# B&R Automation Studio project Assembly_and_ST
Automation Studio 4.5.2.102; technology packages: mappCockpit 5.7.0, mappMotion 5.7.1, mappView 5.7.1

## Configuration Config1

CPU 5PC900.TS77-04, AutomationRuntime D4.52, Build 4.1.2, Vc V4.52.0

### Task classes (Cpu.sw)
```
Cyclic#1 (cycle 800 us, tolerance 0 us):
  ST_Main <- SuperTrak_Module.ST_Main.prg
  MainContro <- Assembly_Module.MainControl.prg
Cyclic#2 (cycle 1600 us, tolerance 0 us):
  AlarmHandl <- Events_handling.AlarmHandling.prg
  AssemblyIn <- Assembly_Module.AssemblyInterface.prg
Cyclic#3 (cycle 9600 us, tolerance 9600 us):
  DisableBra <- Assembly_Module.DisableBrake.prg
  StateMachi <- SuperTrak_Module.StateMachine_SuperTrak.prg
Cyclic#4 (cycle 49600 us, tolerance 49600 us):
  ST_Visu <- SuperTrak_Module.ST_Visu.prg
  EventLogge <- Events_handling.EventLoggerMNG.prg
DataObjects: McAcpSys
Binaries: mvLoader, arcoal, McMechSys, arflatprv, arsvcreg, McProfGen, TCData, McPathXT, mCoWebSc, McAcpSim, McAcpDrv, udbdef, TCLang, Settings, iomap, Config_2, Hierarchy, Config_4, sysconf, ashwac, Config_1, ashwd, asfw, User, arconfig, Config_3, Role, OpcUaMap
Libraries: DataObj, AsArLog, sys_lib, FileIO, AsArProf, AsMem, brsystem, NcGlobal, runtime, astime, AsBrMath, StCom, SuperTrak, AsIecCon, AsBrStr, standard, ArEventLog, AsIODiag, AsGuard, AsTCP, AsIOTime, MpTool, MpBase, McAxGroup, McBase, MpRobotics, MpCnc, MpAxis, McAxis, McProgInt, McPathGen, McPureVAx, McDS402Ax, McAcpPar, McAcpAx, CoTrace, AsZip, asstring, AsARCfg, MpServer, aspciext, asepl, powerlnk, aruser
```

### Hardware
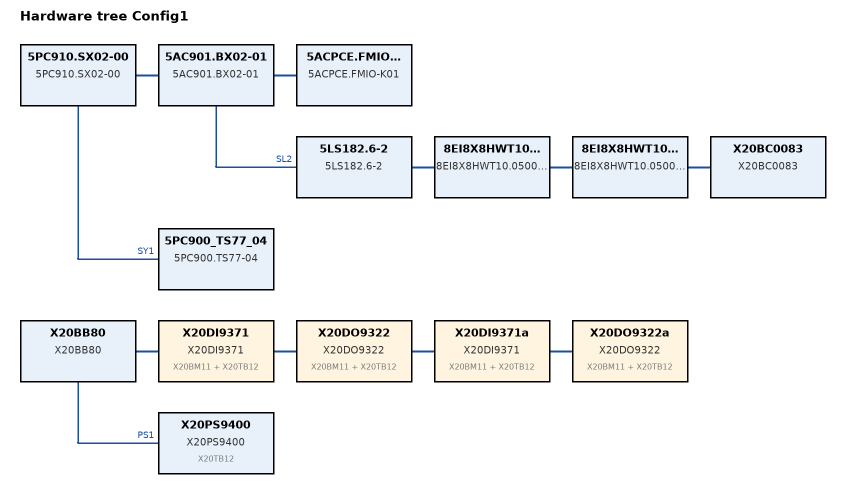
```
5AC901.BX02-01 : 5AC901.BX02-01 v1.1.1.0  [SY -> 5PC910.SX02-00.SY3]
5ACPCE.FMIO-K01 : 5ACPCE.FMIO-K01 v1.0.6.0  [SL -> 5AC901.BX02-01.SL1]
5LS182.6-2 : 5LS182.6-2 v1.3.1.0  [SL -> 5AC901.BX02-01.SL2]
  Connector IF1:
    CycleTime = 800
    Channel1
    ChannelID1 = McAcpBroadcast
    ChannelType1 = OCTET[96]
5PC900_TS77_04 : 5PC900.TS77-04 v2.0.0.0  [SY -> 5PC910.SX02-00.SY1]
  ConfigurationID = ygc_Config1
  UserPartitionSize = 14
  SimulationIPAddress = 192.168.0.101
  UserRamDevice = PCI.2.LS182.SRAM
  UserRamSize = 100000
  RemMemDevice = PCI.2.LS182.SRAM
  RemMemSize = 2048
  PermanentPvSize = 512
  RemanentGlobalPvSize = 512
  VolatileGlobalPvSize = 1026080
  SystemLoggerSize = 614400
  UserLoggerSize = 614400
  TimerDeviceType = EPLX2X
  TimerDevice = 5LS182.6-2.IF1
  TaskClassIdleTime = 800
  Cyclic1Duration = 800
  Cyclic1Tolerance = 0
  Cyclic2Duration = 1600
  Cyclic2Tolerance = 0
  Cyclic3Duration = 9600
  Cyclic3Tolerance = 9600
  Cyclic4Duration = 49600
  Cyclic4Tolerance = 49600
  Cyclic8Duration = 9600
  Cyclic8Tolerance = 0
  FtpUser1
  FtpUsername1 = itq
  FtpUserPassword1 = 7p7ZSnRe8FOUJ14P8lbKBhjsJ4NWIj5puPFWROWS8Pg=
  FtpUserSalt1 = MjfVbkzs
  FTPAccessRight1 = 0
  ActivateOpcUa = 1
  OpcUa_AuthenticationSecurityPolicy_EnableNone = 1
  OpcUa_AuthenticationSecurityPolicy_EnableBasic128Rsa15 = 1
  OpcUaInformationModels_PV_Version = 1
5PC910.SX02-00 : 5PC910.SX02-00 v2.0.0.0
  Connector IF1:
    AssignedOperatingSystem = ARemb
  Connector IF3:
    AssignedOperatingSystem = ARemb
    ActivateDevice = 1
    Mode = Manual
    InternetAddress = 192.168.0.5
    SubnetMask = 255.255.255.0
  Connector IF4:
    AssignedOperatingSystem = ARemb
    ActivateDevice = 1
  Connector IF5:
    AssignedOperatingSystem = ARemb
  Connector IF6:
    AssignedOperatingSystem = ARemb
  Connector IF7:
    AssignedOperatingSystem = ARemb
  Connector IF8:
    AssignedOperatingSystem = ARemb
  Connector IF9:
    AssignedOperatingSystem = ARemb
8EI8X8HWT10.0500-1 : 8EI8X8HWT10.0500-1 v2.2.0.0  [PLK1 -> 5LS182.6-2.IF1 [Cable Type=PowerlinkCable, Length=10, Version=1.0.0.2]; PLK2 -> 8EI8X8HWT10.0500-1a.PLK1 [Cable Type=PowerlinkCable, Length=10, Version=1.0.0.2]]
  DriveConfiguration/Module:
    McAcoposTypeID = AcoposP3TConfig
    ActivateACOPOSSimulationOnPLC = 0
  DriveConfiguration/Encoder/EncoderX41:
    InterfaceType = EnDat
  DriveConfiguration/Encoder/EncoderX42:
    InterfaceType = EnDat
  DriveConfiguration/Encoder/EncoderX43:
    InterfaceType = EnDat
  DriveConfiguration/Channel[1]:
    License = 1
  DriveConfiguration/Channel[1]/RealAxis:
    AxisReference = gAxisQ1
  DriveConfiguration/Channel[1]/RealAxis/MechanicalElements/Gearbox:
    InputIsReadOnly = 1
    Input = 81818
    OutputIsReadOnly = 1
    Output = 1000
  DriveConfiguration/Channel[1]/RealAxis/MechanicalElements/RotaryToLinearTransformation:
    ReferenceDistanceIsReadOnly = 1
    ReferenceDistance = 360
  DriveConfiguration/Channel[1]/RealAxis/Controller:
    ModeIsReadOnly = 1
    Mode = PositionControllerWithTorqueFeedForward
  DriveConfiguration/Channel[1]/RealAxis/Controller/Mode/Position:
    ProportionalGainIsReadOnly = 1
    ProportionalGain = 75.0
    IntegrationTimeIsReadOnly = 1
    IntegrationTime = 0.0
    TotalDelayTime = 0.0004
  DriveConfiguration/Channel[1]/RealAxis/Controller/Mode/Speed:
    ProportionalGainIsReadOnly = 1
    ProportionalGain = 2.0
    IntegrationTimeIsReadOnly = 1
    IntegrationTime = 0.0
    FilterTimeIsReadOnly = 1
    FilterTime = 0.0008
  DriveConfiguration/Channel[1]/RealAxis/Controller/Mode:
    FeedForwardIsReadOnly = 1
    FeedForward = CyclicValueFromAxesGroup
  DriveConfiguration/Channel[1]/RealAxis/Controller/Mode/LoopFilters:
    LoopFilter1 = NotUsed
    LoopFilter2 = NotUsed
    LoopFilter3 = NotUsed
  DriveConfiguration/Channel[1]/RealAxis/Homing:
    Mode = RestorePosition
    RestorePositionVariable = ::MainContro:ResPos[0]
  DriveConfiguration/Channel[1]/RealAxis/StopReaction:
    Quickstop = DecelerationLimit
    DriveError = DecelerationLimit
  DriveConfiguration/Channel[1]/RealAxis/MovementErrorLimits:
    PositionError = 1.0
    VelocityErrorMonitoring = Automatic1
  DriveConfiguration/Channel[1]/RealAxis:
    JerkFilter = Used
  DriveConfiguration/Channel[1]/RealAxis/JerkFilter:
    JerkTime = 0.01
  DriveConfiguration/Channel[1]/RealAxis/DigitalInputs/HomingSwitch:
    Source = NotUsed
    Level = High
  DriveConfiguration/Channel[1]/RealAxis/DigitalInputs/PositiveLimitSwitch:
    Source = NotUsed
    Level = High
  DriveConfiguration/Channel[1]/RealAxis/DigitalInputs/NegativeLimitSwitch:
    Source = NotUsed
    Level = High
  DriveConfiguration/Channel[1]/RealAxis/DigitalInputs/Trigger1:
    Source = X8Trigger1
    Level = High
  DriveConfiguration/Channel[1]/RealAxis/DigitalInputs/Trigger2:
    Source = X8Trigger2
    Level = High
  DriveConfiguration/Channel[1]/RealAxis/DigitalInputs/Quickstop:
    Input = Trigger2
  DriveConfiguration/Channel[1]/RealAxis/Simulation:
    SimulationModeOnPLC = SetValueGeneration
    SimulationModeOnACOPOS = NotUsed
  DriveConfiguration/Channel[2]:
    License = 1
  DriveConfiguration/Channel[2]/RealAxis:
    AxisReference = gAxisQ3
  DriveConfiguration/Channel[2]/RealAxis/MechanicalElements/Gearbox:
    InputIsReadOnly = 1
    Input = 72
    OutputIsReadOnly = 1
    Output = 1
  DriveConfiguration/Channel[2]/RealAxis/MechanicalElements/RotaryToLinearTransformation:
    ReferenceDistanceIsReadOnly = 1
    ReferenceDistance = 360
  DriveConfiguration/Channel[2]/RealAxis/Controller:
    ModeIsReadOnly = 1
    Mode = PositionControllerWithTorqueFeedForward
  DriveConfiguration/Channel[2]/RealAxis/Controller/Mode/Position:
    ProportionalGainIsReadOnly = 1
    ProportionalGain = 50.0
    IntegrationTimeIsReadOnly = 1
    IntegrationTime = 0.0
    TotalDelayTime = 0.0004
  DriveConfiguration/Channel[2]/RealAxis/Controller/Mode/Speed:
    ProportionalGainIsReadOnly = 1
    ProportionalGain = 1.5
    IntegrationTimeIsReadOnly = 1
    IntegrationTime = 0.0
    FilterTimeIsReadOnly = 1
    FilterTime = 0.0008
  DriveConfiguration/Channel[2]/RealAxis/Controller/Mode:
    FeedForwardIsReadOnly = 1
    FeedForward = CyclicValueFromAxesGroup
  DriveConfiguration/Channel[2]/RealAxis/Controller/Mode/LoopFilters:
    LoopFilter1 = NotUsed
    LoopFilter2 = NotUsed
    LoopFilter3 = NotUsed
  DriveConfiguration/Channel[2]/RealAxis/Homing:
    Mode = RestorePosition
    RestorePositionVariable = ::MainContro:ResPos[2]
  DriveConfiguration/Channel[2]/RealAxis/StopReaction:
    Quickstop = DecelerationLimit
    DriveError = DecelerationLimit
  DriveConfiguration/Channel[2]/RealAxis/MovementErrorLimits:
    PositionError = 1.0
    VelocityErrorMonitoring = Automatic1
  DriveConfiguration/Channel[2]/RealAxis:
    JerkFilter = Used
  DriveConfiguration/Channel[2]/RealAxis/JerkFilter:
    JerkTime = 0.01
  DriveConfiguration/Channel[2]/RealAxis/DigitalInputs/HomingSwitch:
    Source = NotUsed
    Level = High
  DriveConfiguration/Channel[2]/RealAxis/DigitalInputs/PositiveLimitSwitch:
    Source = NotUsed
    Level = High
  DriveConfiguration/Channel[2]/RealAxis/DigitalInputs/NegativeLimitSwitch:
    Source = NotUsed
    Level = High
  DriveConfiguration/Channel[2]/RealAxis/DigitalInputs/Trigger1:
    Source = X8Trigger1
    Level = High
  DriveConfiguration/Channel[2]/RealAxis/DigitalInputs/Trigger2:
    Source = X8Trigger2
    Level = High
  DriveConfiguration/Channel[2]/RealAxis/DigitalInputs/Quickstop:
    Input = Trigger2
  DriveConfiguration/Channel[2]/RealAxis/Simulation:
    SimulationModeOnPLC = SetValueGeneration
    SimulationModeOnACOPOS = NotUsed
  DriveConfiguration/Channel[3]:
    License = 1
  DriveConfiguration/Channel[3]/RealAxis:
    AxisReference = gAxisQ5
  DriveConfiguration/Channel[3]/RealAxis/MechanicalElements/Gearbox:
    InputIsReadOnly = 1
    Input = 612
    OutputIsReadOnly = 1
    Output = 10
  DriveConfiguration/Channel[3]/RealAxis/MechanicalElements/RotaryToLinearTransformation:
    ReferenceDistanceIsReadOnly = 1
    ReferenceDistance = 360
  DriveConfiguration/Channel[3]/RealAxis/Controller:
    ModeIsReadOnly = 1
    Mode = PositionControllerWithTorqueFeedForward
  DriveConfiguration/Channel[3]/RealAxis/Controller/Mode/Position:
    ProportionalGainIsReadOnly = 1
    ProportionalGain = 200.0
    IntegrationTimeIsReadOnly = 1
    IntegrationTime = 0.0
    TotalDelayTime = 0.0004
  DriveConfiguration/Channel[3]/RealAxis/Controller/Mode/Speed:
    ProportionalGainIsReadOnly = 1
    ProportionalGain = 1.5
    IntegrationTimeIsReadOnly = 1
    IntegrationTime = 0.0
    FilterTimeIsReadOnly = 1
    FilterTime = 0.0008
  DriveConfiguration/Channel[3]/RealAxis/Controller/Mode:
    FeedForwardIsReadOnly = 1
    FeedForward = CyclicValueFromAxesGroup
  DriveConfiguration/Channel[3]/RealAxis/Controller/Mode/LoopFilters:
    LoopFilter1 = NotUsed
    LoopFilter2 = NotUsed
    LoopFilter3 = NotUsed
  DriveConfiguration/Channel[3]/RealAxis/Homing:
    Mode = RestorePosition
    RestorePositionVariable = ::MainContro:ResPos[4]
  DriveConfiguration/Channel[3]/RealAxis/StopReaction:
    Quickstop = DecelerationLimit
    DriveError = DecelerationLimit
  DriveConfiguration/Channel[3]/RealAxis/MovementErrorLimits:
    PositionError = 1.0
    VelocityErrorMonitoring = Automatic1
  DriveConfiguration/Channel[3]/RealAxis:
    JerkFilter = Used
  DriveConfiguration/Channel[3]/RealAxis/JerkFilter:
    JerkTime = 0.01
  DriveConfiguration/Channel[3]/RealAxis/DigitalInputs/HomingSwitch:
    Source = NotUsed
    Level = High
  DriveConfiguration/Channel[3]/RealAxis/DigitalInputs/PositiveLimitSwitch:
    Source = NotUsed
    Level = High
  DriveConfiguration/Channel[3]/RealAxis/DigitalInputs/NegativeLimitSwitch:
    Source = NotUsed
    Level = High
  DriveConfiguration/Channel[3]/RealAxis/DigitalInputs/Trigger1:
    Source = X8Trigger1
    Level = High
  DriveConfiguration/Channel[3]/RealAxis/DigitalInputs/Trigger2:
    Source = X8Trigger2
    Level = High
  DriveConfiguration/Channel[3]/RealAxis/DigitalInputs/Quickstop:
    Input = Trigger2
  DriveConfiguration/Channel[3]/RealAxis/Simulation:
    SimulationModeOnPLC = SetValueGeneration
    SimulationModeOnACOPOS = NotUsed
8EI8X8HWT10.0500-1a : 8EI8X8HWT10.0500-1 v2.2.0.0  [PLK1 -> 8EI8X8HWT10.0500-1.PLK2 [Cable Type=PowerlinkCable, Length=10, Version=1.0.0.2]; PLK2 -> X20BC0083.PLK1 [Cable Type=PowerlinkCable, Length=10, Version=1.0.0.2]]
  DriveConfiguration/Module:
    McAcoposTypeID = AcoposP3TConfig
    ActivateACOPOSSimulationOnPLC = 0
  DriveConfiguration/Encoder/EncoderX41:
    InterfaceType = EnDat
  DriveConfiguration/Encoder/EncoderX42:
    InterfaceType = EnDat
  DriveConfiguration/Encoder/EncoderX43:
    InterfaceType = EnDat
  DriveConfiguration/Channel[1]:
    License = 1
  DriveConfiguration/Channel[1]/RealAxis:
    AxisReference = gAxisQ2
  DriveConfiguration/Channel[1]/RealAxis/MechanicalElements/Gearbox:
    InputIsReadOnly = 1
    Input = 80
    OutputIsReadOnly = 1
    Output = 1
  DriveConfiguration/Channel[1]/RealAxis/MechanicalElements/RotaryToLinearTransformation:
    ReferenceDistanceIsReadOnly = 1
    ReferenceDistance = 360
  DriveConfiguration/Channel[1]/RealAxis/Controller:
    ModeIsReadOnly = 1
    Mode = PositionControllerWithTorqueFeedForward
  DriveConfiguration/Channel[1]/RealAxis/Controller/Mode/Position:
    ProportionalGainIsReadOnly = 1
    ProportionalGain = 50.0
    IntegrationTimeIsReadOnly = 1
    IntegrationTime = 0.0
    TotalDelayTime = 0.0004
  DriveConfiguration/Channel[1]/RealAxis/Controller/Mode/Speed:
    ProportionalGainIsReadOnly = 1
    ProportionalGain = 2.0
    IntegrationTimeIsReadOnly = 1
    IntegrationTime = 0.0
    FilterTimeIsReadOnly = 1
    FilterTime = 0.0008
  DriveConfiguration/Channel[1]/RealAxis/Controller/Mode:
    FeedForwardIsReadOnly = 1
    FeedForward = CyclicValueFromAxesGroup
  DriveConfiguration/Channel[1]/RealAxis/Controller/Mode/LoopFilters:
    LoopFilter1 = NotUsed
    LoopFilter2 = NotUsed
    LoopFilter3 = NotUsed
  DriveConfiguration/Channel[1]/RealAxis/Homing:
    Mode = RestorePosition
    RestorePositionVariable = ::MainContro:ResPos[1]
  DriveConfiguration/Channel[1]/RealAxis/StopReaction:
    Quickstop = DecelerationLimit
    DriveError = DecelerationLimit
  DriveConfiguration/Channel[1]/RealAxis/MovementErrorLimits:
    PositionError = 1.0
    VelocityErrorMonitoring = Automatic1
  DriveConfiguration/Channel[1]/RealAxis:
    JerkFilter = Used
  DriveConfiguration/Channel[1]/RealAxis/JerkFilter:
    JerkTime = 0.01
  DriveConfiguration/Channel[1]/RealAxis/DigitalInputs/HomingSwitch:
    Source = NotUsed
    Level = High
  DriveConfiguration/Channel[1]/RealAxis/DigitalInputs/PositiveLimitSwitch:
    Source = NotUsed
    Level = High
  DriveConfiguration/Channel[1]/RealAxis/DigitalInputs/NegativeLimitSwitch:
    Source = NotUsed
    Level = High
  DriveConfiguration/Channel[1]/RealAxis/DigitalInputs/Trigger1:
    Source = X8Trigger1
    Level = High
  DriveConfiguration/Channel[1]/RealAxis/DigitalInputs/Trigger2:
    Source = X8Trigger2
    Level = High
  DriveConfiguration/Channel[1]/RealAxis/DigitalInputs/Quickstop:
    Input = Trigger2
  DriveConfiguration/Channel[1]/RealAxis/Simulation:
    SimulationModeOnPLC = SetValueGeneration
    SimulationModeOnACOPOS = NotUsed
  DriveConfiguration/Channel[2]:
    License = 1
  DriveConfiguration/Channel[2]/RealAxis:
    AxisReference = gAxisQ4
  DriveConfiguration/Channel[2]/RealAxis/MechanicalElements/Gearbox:
    InputIsReadOnly = 1
    Input = 612
    OutputIsReadOnly = 1
    Output = 10
  DriveConfiguration/Channel[2]/RealAxis/MechanicalElements/RotaryToLinearTransformation:
    ReferenceDistanceIsReadOnly = 1
    ReferenceDistance = 360
  DriveConfiguration/Channel[2]/RealAxis/Controller:
    ModeIsReadOnly = 1
    Mode = PositionControllerWithTorqueFeedForward
  DriveConfiguration/Channel[2]/RealAxis/Controller/Mode/Position:
    ProportionalGainIsReadOnly = 1
    ProportionalGain = 100.0
    IntegrationTimeIsReadOnly = 1
    IntegrationTime = 0.0
    TotalDelayTime = 0.0004
  DriveConfiguration/Channel[2]/RealAxis/Controller/Mode/Speed:
    ProportionalGainIsReadOnly = 1
    ProportionalGain = 2.0
    IntegrationTimeIsReadOnly = 1
    IntegrationTime = 0.0
    FilterTimeIsReadOnly = 1
    FilterTime = 0.0008
  DriveConfiguration/Channel[2]/RealAxis/Controller/Mode:
    FeedForwardIsReadOnly = 1
    FeedForward = CyclicValueFromAxesGroup
  DriveConfiguration/Channel[2]/RealAxis/Controller/Mode/LoopFilters:
    LoopFilter1 = NotUsed
    LoopFilter2 = NotUsed
    LoopFilter3 = NotUsed
  DriveConfiguration/Channel[2]/RealAxis/Homing:
    Mode = RestorePosition
    RestorePositionVariable = ::MainContro:ResPos[3]
  DriveConfiguration/Channel[2]/RealAxis/StopReaction:
    Quickstop = DecelerationLimit
    DriveError = DecelerationLimit
  DriveConfiguration/Channel[2]/RealAxis/MovementErrorLimits:
    PositionError = 1.0
    VelocityErrorMonitoring = Automatic1
  DriveConfiguration/Channel[2]/RealAxis:
    JerkFilter = Used
  DriveConfiguration/Channel[2]/RealAxis/JerkFilter:
    JerkTime = 0.01
  DriveConfiguration/Channel[2]/RealAxis/DigitalInputs/HomingSwitch:
    Source = NotUsed
    Level = High
  DriveConfiguration/Channel[2]/RealAxis/DigitalInputs/PositiveLimitSwitch:
    Source = NotUsed
    Level = High
  DriveConfiguration/Channel[2]/RealAxis/DigitalInputs/NegativeLimitSwitch:
    Source = NotUsed
    Level = High
  DriveConfiguration/Channel[2]/RealAxis/DigitalInputs/Trigger1:
    Source = X8Trigger1
    Level = High
  DriveConfiguration/Channel[2]/RealAxis/DigitalInputs/Trigger2:
    Source = X8Trigger2
    Level = High
  DriveConfiguration/Channel[2]/RealAxis/DigitalInputs/Quickstop:
    Input = Trigger2
  DriveConfiguration/Channel[2]/RealAxis/Simulation:
    SimulationModeOnPLC = SetValueGeneration
    SimulationModeOnACOPOS = NotUsed
  DriveConfiguration/Channel[3]:
    License = 1
  DriveConfiguration/Channel[3]/RealAxis:
    AxisReference = gAxisQ6
  DriveConfiguration/Channel[3]/RealAxis/MechanicalElements/Gearbox:
    InputIsReadOnly = 1
    Input = 40
    OutputIsReadOnly = 1
    Output = 1
  DriveConfiguration/Channel[3]/RealAxis/MechanicalElements/RotaryToLinearTransformation:
    ReferenceDistanceIsReadOnly = 1
    ReferenceDistance = 360
  DriveConfiguration/Channel[3]/RealAxis/Controller:
    ModeIsReadOnly = 1
    Mode = PositionControllerWithTorqueFeedForward
  DriveConfiguration/Channel[3]/RealAxis/Controller/Mode/Position:
    ProportionalGainIsReadOnly = 1
    ProportionalGain = 200.0
    IntegrationTimeIsReadOnly = 1
    IntegrationTime = 0.0
    TotalDelayTime = 0.0004
  DriveConfiguration/Channel[3]/RealAxis/Controller/Mode/Speed:
    ProportionalGainIsReadOnly = 1
    ProportionalGain = 1.5
    IntegrationTimeIsReadOnly = 1
    IntegrationTime = 0.0
    FilterTimeIsReadOnly = 1
    FilterTime = 0.0008
  DriveConfiguration/Channel[3]/RealAxis/Controller/Mode:
    FeedForwardIsReadOnly = 1
    FeedForward = CyclicValueFromAxesGroup
  DriveConfiguration/Channel[3]/RealAxis/Controller/Mode/LoopFilters:
    LoopFilter1 = NotUsed
    LoopFilter2 = NotUsed
    LoopFilter3 = NotUsed
  DriveConfiguration/Channel[3]/RealAxis/Homing:
    Mode = RestorePosition
    RestorePositionVariable = ::MainContro:ResPos[5]
  DriveConfiguration/Channel[3]/RealAxis/StopReaction:
    Quickstop = DecelerationLimit
    DriveError = DecelerationLimit
  DriveConfiguration/Channel[3]/RealAxis/MovementErrorLimits:
    PositionError = 1.0
    VelocityErrorMonitoring = Automatic1
  DriveConfiguration/Channel[3]/RealAxis:
    JerkFilter = Used
  DriveConfiguration/Channel[3]/RealAxis/JerkFilter:
    JerkTime = 0.01
  DriveConfiguration/Channel[3]/RealAxis/DigitalInputs/HomingSwitch:
    Source = NotUsed
    Level = High
  DriveConfiguration/Channel[3]/RealAxis/DigitalInputs/PositiveLimitSwitch:
    Source = NotUsed
    Level = High
  DriveConfiguration/Channel[3]/RealAxis/DigitalInputs/NegativeLimitSwitch:
    Source = NotUsed
    Level = High
  DriveConfiguration/Channel[3]/RealAxis/DigitalInputs/Trigger1:
    Source = X8Trigger1
    Level = High
  DriveConfiguration/Channel[3]/RealAxis/DigitalInputs/Trigger2:
    Source = X8Trigger2
    Level = High
  DriveConfiguration/Channel[3]/RealAxis/DigitalInputs/Quickstop:
    Input = Trigger2
  DriveConfiguration/Channel[3]/RealAxis/Simulation:
    SimulationModeOnPLC = SetValueGeneration
    SimulationModeOnACOPOS = NotUsed
X20BB80 : X20BB80 v1.0.2.0
X20BC0083 : X20BC0083 v2.7.0.0  [PLK1 -> 8EI8X8HWT10.0500-1a.PLK2 [Cable Type=PowerlinkCable, Length=10, Version=1.0.0.2]; SL -> X20BB80.SL1]
  Supervision = off
X20BM11 : X20BM11 v1.0.0.1  [X2X1 -> X20BB80.IF1]
X20BM11a : X20BM11 v1.0.0.1  [X2X1 -> X20BM11.X2X2]
X20BM11b : X20BM11 v1.0.0.1  [X2X1 -> X20BM11c.X2X2]
X20BM11c : X20BM11 v1.0.0.1  [X2X1 -> X20BM11a.X2X2]
X20DI9371 : X20DI9371 v1.0.2.0  [SS1 -> X20TB12.SS; SL -> X20BM11.SL1]
  Supervision = off
X20DI9371a : X20DI9371 v1.0.2.0  [SS1 -> X20TB12d.SS; SL -> X20BM11c.SL1]
  Supervision = off
X20DO9322 : X20DO9322 v1.0.3.0  [SS1 -> X20TB12b.SS; SL -> X20BM11a.SL1]
  Supervision = off
X20DO9322a : X20DO9322 v1.0.3.0  [SS1 -> X20TB12c.SS; SL -> X20BM11b.SL1]
  Supervision = off
X20PS9400 : X20PS9400 v1.0.2.4  [SS1 -> X20TB12a.SS; PS -> X20BB80.PS1]
  Supervision = off
X20TB12 : X20TB12 v1.0.0.0
X20TB12a : X20TB12 v1.0.0.0
X20TB12b : X20TB12 v1.0.0.0
X20TB12c : X20TB12 v1.0.0.0
X20TB12d : X20TB12 v1.0.0.0
```

### IoMap.iom - 5PC900_TS77_04/IoMap.iom
```iecst
VAR_CONFIG
	::LED_Green AT %QX."X20DO9322".DigitalOutput06;
	::LED_Blue AT %QX."X20DO9322".DigitalOutput07;
	::LED_Red AT %QX."X20DO9322".DigitalOutput08;
	::QA_Actuator_UP AT %QX."X20DO9322".DigitalOutput09;
	::QA_Actuator_DOWN AT %QX."X20DO9322".DigitalOutput10;
	HW_Comau_Gripper AT %QX."X20DO9322a".DigitalOutput01;
	::HW_Assem_RightDoorSensor AT %IX."X20DI9371a".DigitalInput01;
	::HW_Assem_LeftDoorSensor AT %IX."X20DI9371a".DigitalInput02;
	Cyclic#2.::QA_Door_Closed AT %IX."X20DI9371".DigitalInput01;
	ST_LightBarrier_SecurityOut1_R AT %IX."X20DI9371".DigitalInput03;
	ST_LightBarrier_SecurityOut2_R AT %IX."X20DI9371".DigitalInput02;
	::HW_Assem_PelletPresent AT %IX."X20DI9371".DigitalInput06;
	::HW_Assem_PlasticCupsDrawer AT %IX."X20DI9371".DigitalInput05;
	::HW_Assem_PaperCupsDrawer AT %IX."X20DI9371".DigitalInput04;
	::HW_Assem_PlasticLock AT %QX."X20DO9322".DigitalOutput11;
	::HW_Assem_PaperLock AT %QX."X20DO9322".DigitalOutput12;
	::Outfeed_Full AT %IX."X20DI9371a".DigitalInput04;
	::StateMachi:QA_finished AT %IX."X20DI9371a".DigitalInput07;
	::Outfeed_Actuator_BACK AT %QX."X20DO9322".DigitalOutput01;
	::Outfeed_Actuator_FRONT  AT %QX."X20DO9322".DigitalOutput02;
	::Outfeed_Actuator_UP AT %QX."X20DO9322".DigitalOutput03;
	::Outfeed_Actuator_DOWN AT %QX."X20DO9322".DigitalOutput04;
	::Outfeed_LED_Blue  AT %QX."X20DO9322a".DigitalOutput02;
	::Outfeed_LED_Red AT %QX."X20DO9322a".DigitalOutput03;
	::Outfeed_LED_Green AT %QX."X20DO9322a".DigitalOutput04;
END_VAR
```

### Config_3.mechanicalsystem - 5PC900_TS77_04/mappMotion/ComauRacer3/Config_3.mechanicalsystem
```
Element MechSys_ComauRacer3 (Type=mechanicalsystem)
  Type = 6AxesRoboarm
    Subtype = 6AxesRoboarmB
      Description = Standard
        Dimensions:
          TranslationFromBaseToQ1IsReadOnly = 1
          TranslationFromBaseToQ1:
            X = 0.0
            Y = 0.0
            Z = 0.0
          TranslationFromQ1ToQ2IsReadOnly = 1
          TranslationFromQ1ToQ2:
            X = 50.0
            Y = 0.0
            Z = 365.0
          TranslationFromQ2ToQ3IsReadOnly = 1
          TranslationFromQ2ToQ3:
            X = 0.0
            Y = 0.0
            Z = 270.0
          TranslationFromQ3ToQ4IsReadOnly = 1
          TranslationFromQ3ToQ4:
            X = -50.0
            Y = 0.0
            Z = 0.0
          TranslationFromQ4ToQ5IsReadOnly = 1
          TranslationFromQ4ToQ5:
            Z = 305.94
          TranslationFromQ5ToQ6IsReadOnly = 1
          TranslationFromQ5ToQ6:
            Z = 0.0
          TranslationFromQ6ToFlange:
            X = 0.0
            Y = 0.0
            Z = 255
        Offsets:
          JointAxisIsReadOnly = 1
          JointAxis[1] = 0.0
          JointAxis[2] = 0.0
          JointAxis[3] = 0.0
          JointAxis[4] = 0.0
          JointAxis[5] = 0.0
          JointAxis[6] = 0.0
        CountDirections:
          JointAxisIsReadOnly = 1
          JointAxis[1] = Inverse
          JointAxis[2] = Standard
          JointAxis[3] = Inverse
          JointAxis[4] = Inverse
          JointAxis[5] = Standard
          JointAxis[6] = Inverse
      CoordinatesNames = Default
        XCoordinateName = X
        YCoordinateName = Y
        ZCoordinateName = Z
        ACoordinateName = A
        BCoordinateName = B
        CCoordinateName = C
      WireFrameModel = Standard
        Q1ToQ2 = ConnectionLine
          Distance = 0.0
        Q2ToQ3 = ConnectionLine
          Distance = 0.0
        Q3ToQ4 = ConnectionLine
          Distance = 0.0
        Q4ToQ5 = ConnectionLine
          Distance = 0.0
        Q5ToQ6 = ConnectionLine
          Distance = 0.0
        Q6ToFlange = ConnectionLine
          Distance = 0.0
        FlangeToTcp = ConnectionLine
          Distance = 0.0
      DynamicModel = DynParTable
        TableRef
      InternalDynamicModel = Used
        TypeIsReadOnly = 1
        Type = Comau Racer 3
        Row[1]:
          Index = 0
          Value = 4
          Unit = 
          Description = TRF_DYN11D_typ
        Row[2]:
          Index = 1
          Value = 0
          Unit = 
          Description = 
        Row[3]:
          Index = 2
          Value = 0
          Unit = 
          Description = 
        Row[4]:
          Index = 3
          Value = 0.99502
          Unit = kgm^2
          Description = m1*rc1x^2+m1*rc1y^2+Jzz1+(0.0025)*m2+m2*rc2y^2+(0.5)*Jxx2+(-0.5)*Jyy2+(0.5)*Jzz2+(0.0025)*m3+m3*rc3y^2+(0.5)*Jxx3+(-0.5)*Jyy3+(0.5)*Jzz3+(0.0025)*m4+(0.0025)*m5+(0.0025)*m6+(6694.1851)*JDrive1+(-3200)*JDrive2
        Row[5]:
          Index = 4
          Value = 0
          Unit = 
          Description = 
        Row[6]:
          Index = 5
          Value = 0
          Unit = 
          Description = 
        Row[7]:
          Index = 6
          Value = 0
          Unit = 
          Description = 
        Row[8]:
          Index = 7
          Value = -0.0079739
          Unit = kgm
          Description = m2*rc2x
        Row[9]:
          Index = 8
          Value = 0
          Unit = 
          Description = 
        Row[10]:
          Index = 9
          Value = 3.2569
          Unit = kgm
          Description = m2*rc2z+(0.27)*m3+(0.27)*m4+(0.27)*m5+(0.27)*m6
        Row[11]:
          Index = 10
          Value = -0.01529
          Unit = kgm^2
          Description = m2*rc2x*rc2y
        Row[12]:
          Index = 11
          Value = 0.018218
          Unit = kgm^2
          Description = m2*rc2y*rc2z+(0.27)*m3*rc3y
        Row[13]:
          Index = 12
          Value = -0.027
          Unit = kgm^2
          Description = m2*rc2x*rc2z
        Row[14]:
          Index = 13
          Value = 0.23153
          Unit = kgm^2
          Description = m2*rc2x^2+(-0.5)*Jxx2+(0.5)*Jyy2+(0.5)*Jzz2+(3200)*JDrive2
        Row[15]:
          Index = 14
          Value = 0
          Unit = 
          Description = 
        Row[16]:
          Index = 15
          Value = 1.1014
          Unit = kgm^2
          Description = m2*rc2z^2+(0.5)*Jxx2+(0.5)*Jyy2+(-0.5)*Jzz2+(0.0729)*m3+(0.0729)*m4+(0.0729)*m5+(0.0729)*m6+(3200)*JDrive2
        Row[17]:
          Index = 16
          Value = 0
          Unit = 
          Description = 
        Row[18]:
          Index = 17
          Value = 0
          Unit = 
          Description = 
        Row[19]:
          Index = 18
          Value = 0
          Unit = 
          Description = 
        Row[20]:
          Index = 19
          Value = 0
          Unit = 
          Description = 
        Row[21]:
          Index = 20
          Value = -0.32261
          Unit = kgm
          Description = m3*rc3x+(-0.05)*m4+(-0.05)*m5+(-0.05)*m6
        Row[22]:
          Index = 21
          Value = 0
          Unit = 
          Description = 
        Row[23]:
          Index = 22
          Value = 1.1289
          Unit = kgm
          Description = m3*rc3z+m4*rc4z+(0.30594)*m5+(0.30594)*m6
        Row[24]:
          Index = 23
          Value = -0.0059741
          Unit = kgm^2
          Description = m3*rc3x*rc3y
        Row[25]:
          Index = 24
          Value = 0.048102
          Unit = kgm^2
          Description = m3*rc3y*rc3z
        Row[26]:
          Index = 25
          Value = -0.049555
          Unit = kgm^2
          Description = m3*rc3x*rc3z+(-0.05)*m4*rc4z+(-0.015297)*m5+(-0.015297)*m6
        Row[27]:
          Index = 26
          Value = -0.026241
          Unit = kgm^2
          Description = m3*rc3x^2+(-0.5)*Jxx3+(0.5)*Jyy3+(0.5)*Jzz3+(0.0025)*m4+(0.0025)*m5+(0.0025)*m6
        Row[28]:
          Index = 27
          Value = 0
          Unit = 
          Description = 
        Row[29]:
          Index = 28
          Value = 0.21145
          Unit = kgm^2
          Description = m3*rc3z^2+(0.5)*Jxx3+(0.5)*Jyy3+(-0.5)*Jzz3+m4*rc4z^2+(0.5)*Jxx4+(0.5)*Jyy4+(-0.5)*Jzz4+(0.093599)*m5+(0.093599)*m6
        Row[30]:
          Index = 29
          Value = 0
          Unit = 
          Description = 
        Row[31]:
          Index = 30
          Value = 0
          Unit = 
          Description = 
        Row[32]:
          Index = 31
          Value = 0
          Unit = 
          Description = 
        Row[33]:
          Index = 32
          Value = 0
          Unit = 
          Description = 
        Row[34]:
          Index = 33
          Value = -0.0056373
          Unit = kgm
          Description = m4*rc4x
        Row[35]:
          Index = 34
          Value = 0.011806
          Unit = kgm
          Description = m4*rc4y+m5*rc5y
        Row[36]:
          Index = 35
          Value = 0
          Unit = 
          Description = 
        Row[37]:
          Index = 36
          Value = -0.0071612
          Unit = kgm^2
          Description = m4*rc4x*rc4y
        Row[38]:
          Index = 37
          Value = -0.00018934
          Unit = kgm^2
          Description = m4*rc4y*rc4z+(0.30594)*m5*rc5y
        Row[39]:
          Index = 38
          Value = 0.002269
          Unit = kgm^2
          Description = m4*rc4x*rc4z
        Row[40]:
          Index = 39
          Value = -0.0073563
          Unit = kgm^2
          Description = m4*rc4x^2+(-0.5)*Jxx4+(0.5)*Jyy4+(0.5)*Jzz4
        Row[41]:
          Index = 40
          Value = -0.00050442
          Unit = kgm^2
          Description = m4*rc4y^2+(0.5)*Jxx4+(-0.5)*Jyy4+(0.5)*Jzz4+m5*rc5y^2+(0.5)*Jxx5+(-0.5)*Jyy5+(0.5)*Jzz5
        Row[42]:
          Index = 41
          Value = 0
          Unit = 
          Description = 
        Row[43]:
          Index = 42
          Value = 0
          Unit = 
          Description = 
        Row[44]:
          Index = 43
          Value = 0
          Unit = 
          Description = 
        Row[45]:
          Index = 44
          Value = 0
          Unit = 
          Description = 
        Row[46]:
          Index = 45
          Value = 0
          Unit = 
          Description = 
        Row[47]:
          Index = 46
          Value = -0.0030729
          Unit = kgm
          Description = m5*rc5x
        Row[48]:
          Index = 47
          Value = 0
          Unit = 
          Description = 
        Row[49]:
          Index = 48
          Value = 0.0086628
          Unit = kgm
          Description = m5*rc5z+m6*rc6z
        Row[50]:
          Index = 49
          Value = 5.0384e-05
          Unit = kgm^2
          Description = m5*rc5x*rc5y
        Row[51]:
          Index = 50
          Value = 0.004449
          Unit = kgm^2
          Description = m5*rc5y*rc5z
        Row[52]:
          Index = 51
          Value = 0.00094987
          Unit = kgm^2
          Description = m5*rc5x*rc5z
        Row[53]:
          Index = 52
          Value = -0.0039698
          Unit = kgm^2
          Description = m5*rc5x^2+(-0.5)*Jxx5+(0.5)*Jyy5+(0.5)*Jzz5
        Row[54]:
          Index = 53
          Value = 0
          Unit = 
          Description = 
        Row[55]:
          Index = 54
          Value = -0.0023413
          Unit = kgm^2
          Description = m5*rc5z^2+(0.5)*Jxx5+(0.5)*Jyy5+(-0.5)*Jzz5+m6*rc6z^2+(0.5)*Jxx6+(0.5)*Jyy6+(-0.5)*Jzz6
        Row[56]:
          Index = 55
          Value = 0
          Unit = 
          Description = 
        Row[57]:
          Index = 56
          Value = 0
          Unit = 
          Description = 
        Row[58]:
          Index = 57
          Value = 0
          Unit = 
          Description = 
        Row[59]:
          Index = 58
          Value = 0
          Unit = 
          Description = 
        Row[60]:
          Index = 59
          Value = 0.00052765
          Unit = kgm
          Description = m6*rc6x
        Row[61]:
          Index = 60
          Value = -0.0030867
          Unit = kgm
          Description = m6*rc6y
        Row[62]:
          Index = 61
          Value = 0
          Unit = 
          Description = 
        Row[63]:
          Index = 62
          Value = 5.0962e-05
          Unit = kgm^2
          Description = m6*rc6x*rc6y
        Row[64]:
          Index = 63
          Value = -0.0015762
          Unit = kgm^2
          Description = m6*rc6y*rc6z
        Row[65]:
          Index = 64
          Value = 0.0005846
          Unit = kgm^2
          Description = m6*rc6x*rc6z
        Row[66]:
          Index = 65
          Value = 0.00067399
          Unit = kgm^2
          Description = m6*rc6x^2+(-0.5)*Jxx6+(0.5)*Jyy6+(0.5)*Jzz6
        Row[67]:
          Index = 66
          Value = 0.0013929
          Unit = kgm^2
          Description = m6*rc6y^2+(0.5)*Jxx6+(-0.5)*Jyy6+(0.5)*Jzz6
        Row[68]:
          Index = 67
          Value = 0
          Unit = 
          Description = 
        Row[69]:
          Index = 68
          Value = 0
          Unit = 
          Description = 
        Row[70]:
          Index = 69
          Value = 0
          Unit = 
          Description = 
        Row[71]:
          Index = 70
          Value = 0
          Unit = 
          Description = 
        Row[72]:
          Index = 71
          Value = 0
          Unit = 
          Description = mTool
        Row[73]:
          Index = 72
          Value = 0
          Unit = 
          Description = mTool*rcToolx
        Row[74]:
          Index = 73
          Value = 0
          Unit = 
          Description = mTool*rcTooly
        Row[75]:
          Index = 74
          Value = 0
          Unit = 
          Description = mTool*rcToolz
        Row[76]:
          Index = 75
          Value = 0
          Unit = 
          Description = mTool*rcToolx*rcTooly
        Row[77]:
          Index = 76
          Value = 0
          Unit = 
          Description = mTool*rcTooly*rcToolz
        Row[78]:
          Index = 77
          Value = 0
          Unit = 
          Description = mTool*rcToolx*rcToolz
        Row[79]:
          Index = 78
          Value = 0
          Unit = 
          Description = mTool*rcToolx^2
        Row[80]:
          Index = 79
          Value = 0
          Unit = 
          Description = mTool*rcTooly^2
        Row[81]:
          Index = 80
          Value = 0
          Unit = 
          Description = mTool*rcToolz^2
        Row[82]:
          Index = 81
          Value = 0
          Unit = 
          Description = JxxTool
        Row[83]:
          Index = 82
          Value = 0
          Unit = 
          Description = JyyTool
        Row[84]:
          Index = 83
          Value = 0
          Unit = 
          Description = JzzTool
        Row[85]:
          Index = 84
          Value = 0
          Unit = 
          Description = 
        Row[86]:
          Index = 85
          Value = 0
          Unit = 
          Description = 
        Row[87]:
          Index = 86
          Value = 9.8824e-05
          Unit = kgm^2
          Description = JDrive3
        Row[88]:
          Index = 87
          Value = 5.2689e-05
          Unit = kgm^2
          Description = JDrive4
        Row[89]:
          Index = 88
          Value = 5.129e-05
          Unit = kgm^2
          Description = JDrive5
        Row[90]:
          Index = 89
          Value = 5.2318e-05
          Unit = kgm^2
          Description = JDrive6
        Row[91]:
          Index = 90
          Value = 4.1946
          Unit = Nms
          Description = dV1
        Row[92]:
          Index = 91
          Value = 7.0888
          Unit = Nms
          Description = dV2
        Row[93]:
          Index = 92
          Value = 3.1195
          Unit = Nms
          Description = dV3
        Row[94]:
          Index = 93
          Value = 1.481
          Unit = Nms
          Description = dV4
        Row[95]:
          Index = 94
          Value = 1.1989
          Unit = Nms
          Description = dV5
        Row[96]:
          Index = 95
          Value = 0.67577
          Unit = Nms
          Description = dV6
        Row[97]:
          Index = 96
          Value = 25.5954
          Unit = Nm
          Description = dC1
        Row[98]:
          Index = 97
          Value = 14.3239
          Unit = Nm
          Description = dC2
        Row[99]:
          Index = 98
          Value = 7.6123
          Unit = Nm
          Description = dC3
        Row[100]:
          Index = 99
          Value = 7.9035
          Unit = Nm
          Description = dC4
        Row[101]:
          Index = 100
          Value = 3.5858
          Unit = Nm
          Description = dC5
        Row[102]:
          Index = 101
          Value = 5.2501
          Unit = Nm
          Description = dC6
      Couplings:
        LinearCoupling[1]:
          SourceAxisIsReadOnly = 1
          SourceAxis = 5
          SourceAxisUnitsIsReadOnly = 1
          SourceAxisUnits = 1.0
          TargetJointAxisIsReadOnly = 1
          TargetJointAxis = 6
          TargetJointAxisUnitsIsReadOnly = 1
          TargetJointAxisUnits = 0.02
      JointAxesPositionLimits:
        JointAxis[1] = ConfigureJointAxesLimits
          LowerLimitMin = -170.0
          UpperLimitMax = 170.0
          LowerLimit = -170.0
          UpperLimit = 170.0
        JointAxis[2] = ConfigureJointAxesLimits
          LowerLimitMin = -95.0
          UpperLimitMax = 135.0
          LowerLimit = -95.0
          UpperLimit = 135.0
        JointAxis[3] = ConfigureJointAxesLimits
          LowerLimitMin = -155.0
          UpperLimitMax = 90.0
          LowerLimit = -155.0
          UpperLimit = 90.0
        JointAxis[4] = ConfigureJointAxesLimits
          LowerLimitMin = -200.0
          UpperLimitMax = 200.0
          LowerLimit = -200.0
          UpperLimit = 200.0
        JointAxis[5] = ConfigureJointAxesLimits
          LowerLimitMin = -125.0
          UpperLimitMax = 125.0
          LowerLimit = -125.0
          UpperLimit = 125.0
        JointAxis[6] = ConfigureJointAxesLimits
          LowerLimitMin = -2700.0
          UpperLimitMax = 2700.0
          LowerLimit = -2700.0
          UpperLimit = 2700.0
```

### Config_4.axesgroupfeature - 5PC900_TS77_04/mappMotion/ComauRacer3/Config_4.axesgroupfeature
```
Element Feature_Programs (Type=axesgroupfeature)
  Type = Program
    ModalDataBehaviour = UseAxesGroupSettings
    InitialSettings:
      InterpolationTypes = LinearRapid
      PositionCoordinates = Absolute
      CircleCoordinates = Relative
      JACS_ACSProgramming = JACS
      ContourConnection = Inactive
      ProgrammingUnits = UseAxesGroupSettings
      Feedrates:
        FeedCharacteristic = StandardCharacteristic
        FeedType = Feedrate
        FeedrateValue = 0.0
        InverseFeedrateValue = 0.0
        FeedratePerRevValue = 0.0
    DefaultLanguage = BRGCode
    Location = Default
      FileDevice = CNC_PrgDir
Element Feature_FeedForward (Type=axesgroupfeature)
  Type = FeedForward
    Mode = ComputeAndTransmit
    RiseTime = 0.25
Element Feature_Jogging (Type=axesgroupfeature)
  Type = Jogging
```

## Logical view

Binary libraries used (declarations not repeated): operator, runtime, astime, AsIecCon, DataObj, AsArLog, sys_lib, FileIO, AsArProf, AsMem, brsystem, NcGlobal, AsBrMath, StCom 5.03.0, SuperTrak, AsBrStr, standard, ArEventLog, AsIODiag, AsGuard, AsTCP, AsIOTime, MpBase, CoTrace 5.07.0, AsZip, asstring, AsARCfg, MpServer 5.07.0, MpTool, MpRobotics, MpCnc 5.07.1, MpAxis 5.07.1, McProgInt 5.07.1, McPathGen, McPureVAx, McDS402Ax 5.07.1, McAxGroup 5.07.1, McAxis, McAcpAx 5.07.1, McAcpPar 5.07.1, McBase 5.07.1

### Package Logical/Libraries - Global libraries

### Global_Constants.var
```iecst
(* ******************************************************************************** *)
VAR CONSTANT
	CONFIG_SUPERTRAK_LENGTH : DINT := 6020; (* Supertrak Length for Simulation *)
	CONFIG_SECTION_LENGTH : DINT := 1000; (* Section Length in mm *)
END_VAR
(* ******************************************************************************** *)
(* ******************************************************************************** *)
(* Lifebit Timeout *)
(* ******************************************************************************** *)
VAR CONSTANT
	LIFEBIT_TIMEOUT : TIME := T#5000ms;
	SUPERTRAK_MAX_COMMANDS_DIV_8_M1 : USINT := 5; (*M1=Minus one*)
	SUPERTRAK_MAX_IOS : USINT := 128;
	SUPERTRAK_MAX_IOS_DIV_8_M1 : USINT := 15; (*M1=Minus one*)
	SUPERTRAK_MAX_SECTIONS : USINT := 6;
	SUPERTRAK_MAX_SHUTTLES : USINT := 16;
	SUPERTRAK_MAX_SECTIONS_MINUS_1 : USINT := 5;
	SUPERTRAK_MAX_TARGETS : USINT := 128;
	SUPERTRAK_MAX_TARGETS_MINUS_1 : USINT := 127;
	SUPERTRAK_MAX_TARGETS_DIV_4_M1 : USINT := 31; (*M1=Minus one*)
	SUPERTRAK_SHUTTLES : USINT := 6;
	SUPERTRAK_SECTIONS : USINT := 6;
	SUPERTRAK_TARGETS : USINT := 8;
	SUPERTRAK_MAX_COMMANDS_MINUS_1 : USINT := 47;
	SUPERTRAK_SKILLS : USINT := 9;
END_VAR
(* SuperTrak Constants *)
(* ******************************************************************************** *)
VAR CONSTANT
	SUPERTRAK_MAX_COMMANDS : USINT := 48;
END_VAR
```

### Global.var
```iecst
VAR
	Life_Bit_Ignore : BOOL := TRUE; (*Flag for simulation without life bit acknowledge from the MES*)
	TON_AssemblyLifeBit : TON;
	Ack : USINT;
	TON_SuperTrakLifeBit : TON;
END_VAR
```

### Program Logical/Assembly_Module/AssemblyInterface (IEC)

#### Main.st
```iecst
PROGRAM _INIT

END_PROGRAM

PROGRAM _CYCLIC

(******************************************************************************************************************)

	(*********************)
	//(*INPUT INTERFACE*)//
	(*********************)

	//(*HARDWARE INPUT VARIABLES*)//

	(*Angles of the Comau assigned from AS Library for Comau*)
	(*they will allway come from the "Hardware" side because there is no transformation in the robot in the Digital tween*)

	Comau_Joint_1_Angle := Mp_Comau.Info.JointAxisPosition[0];
	Comau_Joint_2_Angle := Mp_Comau.Info.JointAxisPosition[1];
	Comau_Joint_3_Angle := Mp_Comau.Info.JointAxisPosition[2];
	Comau_Joint_4_Angle := Mp_Comau.Info.JointAxisPosition[3];
	Comau_Joint_5_Angle := Mp_Comau.Info.JointAxisPosition[4];
	Comau_Joint_6_Angle := Mp_Comau.Info.JointAxisPosition[5];

	(*Signal to detect if the gripper has already grabbed an object coming from the hardware*)

	IF NOT DiagCpuIsSimulated() THEN

	//	Comau_IsGrabbing 					:= HW_Comau_IsGrabbing; we don't have this signal (it does not exist)

		Assem_LeftDoorSensor 				:= HW_Assem_LeftDoorSensor;
		Assem_RightDoorSensor 				:= HW_Assem_RightDoorSensor;

		Assem_PelletPresent					:= HW_Assem_PelletPresent;

		Assem_PlasticCupsDrawer				:= HW_Assem_PlasticCupsDrawer;
		Assem_PaperCupsDrawer				:= HW_Assem_PaperCupsDrawer;

	END_IF

	//(*SIMULATION INPUT VARIABLES*)//

	(*Signal to detect if the gripper has already grabbed an object coming from Industrial Physics*)

	IF DiagCpuIsSimulated() THEN
		Comau_IsGrabbing :=  SimInputs.Gripper01_VACUUM;

//		Assem_PlasticRightDoor_Sensor 	:= SimInputs.DT_Assem_PlasticRightDoor_Sensor;
//		Assem_PlasticLeftDoor_Sensor	:= SimInputs.DT_Assem_PlasticLeftDoor_Sensor;

//		Assem_PaperRightDoor_Sensor 	:= SimInputs.DT_Assem_PaperRightDoor_Sensor;
//		Assem_PaperLeftDoor_Sensor		:= SimInputs.DT_Assem_PaperLeftDoor_Sensor;
	END_IF

	//End of the Input variables Interface
(******************************************************************************************************************)

	(*********************)
	//(*OUTPUT INTERFACE*)//
	(*********************)

	//(*HARDWARE OUTPUT VARIABLES*)//

	(*Here are defined the ouput variables for the hardware*)
	(* They only will work iF the simulation mode is no active*)

	IF NOT DiagCpuIsSimulated() THEN

		HW_Comau_Gripper 		:= Comau_Gripper;

		HW_Assem_PlasticLock 	:= Assem_PlasticLock;
		HW_Assem_PlasticLock 	:= Assem_PlasticLock;

	END_IF

	//(*SIMULATION OUTPUT VARIABLES*)//

	(*Here are defined all the outputs that go to Industrial physics and to the Hardware*)
	(*they are allway assigned because the simulation MUST always work*)

	(*Angles of the Comau assigned to Industrial Physics variables*)

	SimOutputs.Comau_Link101_TGT_POS := LREAL_TO_REAL(Comau_Joint_1_Angle);
	SimOutputs.Comau_Link201_TGT_POS := LREAL_TO_REAL(Comau_Joint_2_Angle);
	SimOutputs.Comau_Link301_TGT_POS := LREAL_TO_REAL(Comau_Joint_3_Angle);
	SimOutputs.Comau_Link401_TGT_POS := LREAL_TO_REAL(Comau_Joint_4_Angle);
	SimOutputs.Comau_Link501_TGT_POS := LREAL_TO_REAL(Comau_Joint_5_Angle);
	SimOutputs.Comau_Link601_TGT_POS := LREAL_TO_REAL(Comau_Joint_6_Angle);

	(*Security sensor variables assigned to an Industrial Physics variable*)

	SimOutputs.PlasticCupDrawer01_Assem := Assem_PlasticCupsDrawer;
	SimOutputs.PaperCupDrawer01_Assem := Assem_PaperCupsDrawer;

	(*Grpper of the Comau assigned to an Industrial Physics variable*)

	SimOutputs.Gripper01_GRIP := Comau_Gripper;

	//End of the Output variables Interface
(*****************************************************************************************************************)

END_PROGRAM

PROGRAM _EXIT

END_PROGRAM
```

### Program Logical/Assembly_Module/MainControl (IEC)

#### Cyclic.st
```iecst
PROGRAM _CYCLIC

	(*************************************************************************************************)
	(* General Actions Call*)
	(*************************************************************************************************)

	SuperState;
	StateMachine;

	(*************************************************************************************************)
	(* Skills Actions Call*)
	(*************************************************************************************************)

	goHome;
	provideCup;
	providePellet;

END_PROGRAM
```

#### Init.st
```iecst
PROGRAM _INIT

	Mp_Joint[0].Enable := TRUE;
	Mp_Joint[0].MpLink := ADR(gAxisQ1);
	Mp_Joint[0].Parameters := ADR(Mp_JointParameters[0]);
	Mp_JointParameters[0].Homing.Mode := mcHOMING_DEFAULT;

	Mp_Joint[1].Enable := TRUE;
	Mp_Joint[1].MpLink := ADR(gAxisQ2);
	Mp_Joint[1].Parameters := ADR(Mp_JointParameters[1]);
	Mp_JointParameters[1].Homing.Mode := mcHOMING_DEFAULT;

	Mp_Joint[2].Enable := TRUE;
	Mp_Joint[2].MpLink := ADR(gAxisQ3);
	Mp_Joint[2].Parameters := ADR(Mp_JointParameters[2]);
	Mp_JointParameters[2].Homing.Mode := mcHOMING_DEFAULT;

	Mp_Joint[3].Enable := TRUE;
	Mp_Joint[3].MpLink := ADR(gAxisQ4);
	Mp_Joint[3].Parameters := ADR(Mp_JointParameters[3]);
	Mp_JointParameters[3].Homing.Mode := mcHOMING_DEFAULT;

	Mp_Joint[4].Enable := TRUE;
	Mp_Joint[4].MpLink := ADR(gAxisQ5);
	Mp_Joint[4].Parameters := ADR(Mp_JointParameters[4]);
	Mp_JointParameters[4].Homing.Mode := mcHOMING_DEFAULT;

	Mp_Joint[5].Enable := TRUE;
	Mp_Joint[5].MpLink := ADR(gAxisQ6);
	Mp_Joint[5].Parameters := ADR(Mp_JointParameters[5]);
	Mp_JointParameters[5].Homing.Mode := mcHOMING_DEFAULT;

	Mp_Comau.MpLink := ADR(gComauRacer3);
	Mp_Comau.Enable := TRUE;
	Mp_Comau.Parameters := ADR(Mp_Parameters);

	Mp_Comau.Override := 100.0;
	Mp_Parameters.CoordSystem := 4;

	//SKILS names initialization
	gAssemblyModule.skill.goHome.name := 'goHome';
	gAssemblyModule.skill.provideCup.name := 'provideCup';
	gAssemblyModule.skill.providePellet.name := 'providePellet';

	provideCup_Case := CUP_SUPPLY_DECISION_CASE;
	providePellet_Case := PELLET_SUPPLY_DECISION_CASE;

	// adapt supply INIT positions
	Paper_Cup_Supply_Position := PAPER_CUP_INIT_POSITION;
	Plastic_Cup_Supply_Position := PLASTIC_CUP_INIT_POSITION;

	//Safe-Positions INIT
	Plastic_Cup_Safe_Pos := PLASTIC_CUP_INIT_POSITION;
	Paper_Cup_Safe_Pos := PAPER_CUP_INIT_POSITION;

	// define "above" positions dependent on the referred position
	Paper_Cup_Supply_Above_Pos := Paper_Cup_Supply_Position;
	Plastic_Cup_Supply_Above_Pos := Plastic_Cup_Supply_Position;
	Supertrak_Above_Position := Supertrak_Position;
	Small_Pellet_Supply_Pos_Before := Small_Pellet_Supply_Pos;

	Supertrak_Above_Position[2] := Supertrak_Above_Position[2] + 70;

	Paper_Cup_Supply_Above_Pos[2] := Paper_Cup_Supply_Position[2] + 60;
	Plastic_Cup_Supply_Above_Pos[2] := Paper_Cup_Supply_Position[2] + 60;

	Small_Pellet_Supply_Pos_Before[2] := Small_Pellet_Supply_Pos_Before[2] +65;

	Plastic_Cup_Safe_Pos[0] := 0;
	Plastic_Cup_Safe_Pos[1] := PAPER_CUP_INIT_POSITION[1]*(-1) - 200;
	Plastic_Cup_Safe_Pos[2] := Supertrak_Above_Position[2];

	Paper_Cup_Safe_Pos[0] := 0;
	Paper_Cup_Safe_Pos[1] := PAPER_CUP_INIT_POSITION[1] +200;
	Paper_Cup_Safe_Pos[2] := Supertrak_Above_Position[2];

	Assem_PaperLock := TRUE;
	Assem_PlasticLock := TRUE;
	Refill_Done := FALSE;
	Plastic_RefillDone := TRUE;
	Paper_RefillDone := TRUE;

END_PROGRAM
```

#### SuperState.st
```iecst
ACTION SuperState:

(*************************************************************************************************)
(*Lifebit*)
(*************************************************************************************************)
	(* If the flag is set the code can be simulated wothout the lifebit taken into account *)
	IF NOT Life_Bit_Ignore THEN

		IF gAssemblyModule.lifeBit.lifeBitAck THEN

			gAssemblyModule.lifeBit.lifeBitAck := FALSE;
			TON_AssemblyLifeBit(IN := FALSE);
			TON_AssemblyLifeBit(IN := TRUE, PT := LIFEBIT_TIMEOUT);

		ELSIF NOT gAssemblyModule.lifeBit.lifeBitAck AND

			TON_AssemblyLifeBit.ET >= LIFEBIT_TIMEOUT THEN
			Event_Code := 104;
			EventLog.Commands.WriteUserEvent := TRUE;
			TON_AssemblyLifeBit(IN := FALSE);

		END_IF;

		TON_AssemblyLifeBit();

	END_IF;

	(*************************************************************************************************)

	//call axis and comau configuration FBs
	FOR i:=0 TO 5 DO
		Mp_Joint[i]();
	END_FOR

	Mp_Comau();

	//Push Emergency Button Case (only way to know if its pressed)
	IF NOT Mp_Comau.Info.ReadyToPowerOn THEN
		Event_Code := 200;
		EventLog.Commands.WriteUserEvent := TRUE;
	END_IF

	//MAINTENANCE REQUESTED
	//First it will finish the completing and then it will enter in this mode
	IF (gAssemblyModule.skill.goHome.state.stateMachine.operationalState = COMPLETING OR
		gAssemblyModule.skill.provideCup.state.stateMachine.operationalState = COMPLETING OR
		gAssemblyModule.skill.providePellet.state.stateMachine.operationalState = COMPLETING) AND
		Maintenance_Requested THEN

		Stopped_Case := MAINTENANCE_STOPPED;
		Maintenance_Requested := FALSE;
		gAssemblyModule.state.stateMachine.stateTransition.stop := TRUE;

		//generate warning message
		Event_Code := 200;
		EventLog.Commands.WriteUserEvent := TRUE;

	END_IF

	//Illegal position in the cup tray, should be AND (still to find out the error code)
	IF (Mp_Comau.Error OR Mp_Comau.StatusID = 1111111)
		AND (gAssemblyModule.skill.provideCup.state.stateMachine.operationalState = RUNNING) THEN
		Event_Code := 101;
		EventLog.Commands.WriteUserEvent := TRUE;
	END_IF

	//Error in Homing Procedure
	IF (Mp_Comau.Error OR Mp_Comau.StatusID = -1067211008) THEN
		Event_Code := 131;
		EventLog.Commands.WriteUserEvent := TRUE;
	END_IF

	//Errors of illegally opening doors or drawers
	IF gAssemblyModule.state.stateMachine.operationalState <> ABORTED AND
		NOT Assem_IgnoreSafetySensors THEN

		IF NOT Assem_LeftDoorSensor OR NOT Assem_RightDoorSensor THEN
			Event_Code := 140;
			EventLog.Commands.WriteUserEvent := TRUE;
		END_IF

		IF gAssemblyModule.state.stateMachine.operationalState <> HELD OR
			gAssemblyModule.state.stateMachine.operationalState <> UNHOLDING THEN

			IF TON_DrawerAlarm.Q AND NOT Assem_PlasticCupsDrawer THEN
				Event_Code := 144;
				EventLog.Commands.WriteUserEvent := TRUE;
			END_IF;

			IF TON_DrawerAlarm.Q AND NOT Assem_PaperCupsDrawer THEN
				Event_Code := 145;
				EventLog.Commands.WriteUserEvent := TRUE;
			END_IF;
		END_IF;

	END_IF

	TON_DrawerAlarm(IN := Assem_PlasticCupsDrawer OR Assem_PaperCupsDrawer, PT := T#1s);

END_ACTION
```

#### Program Logical/Assembly_Module/MainControl/Functions

##### F_Plastic_Update_Positions.st
```iecst
FUNCTION F_Plastic_Update_Positions

	IF (y_counter_plastic = 0) AND (x_counter_plastic < 4) THEN //this raw has only 5 cups

		x_counter_plastic := x_counter_plastic + 1;
		Plastic_Cup_Supply_Above_Pos[0] := PLASTIC_CUP_INIT_POSITION [0] - DIST_X_PLASTIC_CENTR_SAME_ROW * x_counter_plastic * COS(PLASTIC_TRAY_ORIENTATION);
		Plastic_Cup_Supply_Position[0] := PLASTIC_CUP_INIT_POSITION [0] - DIST_X_PLASTIC_CENTR_SAME_ROW * x_counter_plastic * COS(PLASTIC_TRAY_ORIENTATION);
		Plastic_Cup_Supply_Above_Pos[1] := PLASTIC_CUP_INIT_POSITION [1] - DIST_Y_PLASTIC_CENTR * y_counter_plastic;
		Plastic_Cup_Supply_Position[1] := PLASTIC_CUP_INIT_POSITION [1] - DIST_Y_PLASTIC_CENTR * y_counter_plastic;
		Plastic_Cups_Remaining := Plastic_Cups_Remaining -1;
		RETURN;
	ELSIF (y_counter_plastic = 0) AND (x_counter_plastic = 4) THEN //this raw has only 5 cups last case
		x_counter_plastic := 0;
		y_counter_plastic := 1;
		Plastic_Cup_Supply_Above_Pos[0] := PLASTIC_CUP_INIT_POSITION [0] - DIST_X_PLASTIC_CENTR_SAME_ROW * x_counter_plastic * COS(PLASTIC_TRAY_ORIENTATION) -50 +200;
		Plastic_Cup_Supply_Position[0] := PLASTIC_CUP_INIT_POSITION [0] - DIST_X_PLASTIC_CENTR_SAME_ROW * x_counter_plastic * COS(PLASTIC_TRAY_ORIENTATION) -50 +200;
		Plastic_Cup_Supply_Above_Pos[1] := PLASTIC_CUP_INIT_POSITION [1] - DIST_Y_PLASTIC_CENTR * y_counter_plastic;
		Plastic_Cup_Supply_Position[1] := PLASTIC_CUP_INIT_POSITION [1] - DIST_Y_PLASTIC_CENTR * y_counter_plastic;
		Plastic_Cups_Remaining := Plastic_Cups_Remaining -1;
		RETURN;
	END_IF

	IF (y_counter_plastic = 1) AND (x_counter_plastic < 7) THEN

		x_counter_plastic := x_counter_plastic + 1;
		Plastic_Cup_Supply_Above_Pos[0] := PLASTIC_CUP_INIT_POSITION [0] - DIST_X_PLASTIC_CENTR_SAME_ROW * x_counter_plastic * COS(PLASTIC_TRAY_ORIENTATION) -50 +200;
		Plastic_Cup_Supply_Position[0] := PLASTIC_CUP_INIT_POSITION [0] - DIST_X_PLASTIC_CENTR_SAME_ROW * x_counter_plastic * COS(PLASTIC_TRAY_ORIENTATION) -50 +200;
		Plastic_Cup_Supply_Above_Pos[1] := PLASTIC_CUP_INIT_POSITION [1] - DIST_Y_PLASTIC_CENTR * y_counter_plastic;
		Plastic_Cup_Supply_Position[1] := PLASTIC_CUP_INIT_POSITION [1] - DIST_Y_PLASTIC_CENTR * y_counter_plastic;
		Plastic_Cups_Remaining := Plastic_Cups_Remaining -1;
		RETURN;
	ELSIF (y_counter_plastic = 1) AND (x_counter_plastic = 7) THEN //this raw has only 5 cups last case
		x_counter_plastic := 0;
		y_counter_plastic := 2;
		Plastic_Cup_Supply_Above_Pos[0] := PLASTIC_CUP_INIT_POSITION [0] - DIST_X_PLASTIC_CENTR_SAME_ROW * x_counter_plastic * COS(PLASTIC_TRAY_ORIENTATION) +200;
		Plastic_Cup_Supply_Position[0] := PLASTIC_CUP_INIT_POSITION [0] - DIST_X_PLASTIC_CENTR_SAME_ROW * x_counter_plastic * COS(PLASTIC_TRAY_ORIENTATION) +200;
		Plastic_Cup_Supply_Above_Pos[1] := PLASTIC_CUP_INIT_POSITION [1] - DIST_Y_PLASTIC_CENTR * y_counter_plastic;
		Plastic_Cup_Supply_Position[1] := PLASTIC_CUP_INIT_POSITION [1] - DIST_Y_PLASTIC_CENTR * y_counter_plastic;
		Plastic_Cups_Remaining := Plastic_Cups_Remaining -1;
		RETURN;
	END_IF

	IF (y_counter_plastic = 2) AND (x_counter_plastic < 8) THEN

		x_counter_plastic := x_counter_plastic + 1;
		Plastic_Cup_Supply_Above_Pos[0] := PLASTIC_CUP_INIT_POSITION [0] - DIST_X_PLASTIC_CENTR_SAME_ROW * x_counter_plastic * COS(PLASTIC_TRAY_ORIENTATION) +200;
		Plastic_Cup_Supply_Position[0] := PLASTIC_CUP_INIT_POSITION [0] - DIST_X_PLASTIC_CENTR_SAME_ROW * x_counter_plastic * COS(PLASTIC_TRAY_ORIENTATION) +200;
		Plastic_Cup_Supply_Above_Pos[1] := PLASTIC_CUP_INIT_POSITION [1] - DIST_Y_PLASTIC_CENTR * y_counter_plastic;
		Plastic_Cup_Supply_Position[1] := PLASTIC_CUP_INIT_POSITION [1] - DIST_Y_PLASTIC_CENTR * y_counter_plastic;
		Plastic_Cups_Remaining := Plastic_Cups_Remaining -1;
		RETURN;
	ELSIF (y_counter_plastic = 2) AND (x_counter_plastic = 8) THEN //this raw has only 5 cups last case
		x_counter_plastic := 0;
		y_counter_plastic := 3;
		Plastic_Cup_Supply_Above_Pos[0] := PLASTIC_CUP_INIT_POSITION [0] - DIST_X_PLASTIC_CENTR_SAME_ROW * x_counter_plastic * COS(PLASTIC_TRAY_ORIENTATION) -50 +200;
		Plastic_Cup_Supply_Position[0] := PLASTIC_CUP_INIT_POSITION [0] - DIST_X_PLASTIC_CENTR_SAME_ROW * x_counter_plastic * COS(PLASTIC_TRAY_ORIENTATION) -50 +200;
		Plastic_Cup_Supply_Above_Pos[1] := PLASTIC_CUP_INIT_POSITION [1] - DIST_Y_PLASTIC_CENTR * y_counter_plastic;
		Plastic_Cup_Supply_Position[1] := PLASTIC_CUP_INIT_POSITION [1] - DIST_Y_PLASTIC_CENTR * y_counter_plastic;
		Plastic_Cups_Remaining := Plastic_Cups_Remaining -1;
		RETURN;
	END_IF

	IF (y_counter_plastic = 3) AND (x_counter_plastic < 7) THEN

		x_counter_plastic := x_counter_plastic + 1;
		Plastic_Cup_Supply_Above_Pos[0] := PLASTIC_CUP_INIT_POSITION [0] - DIST_X_PLASTIC_CENTR_SAME_ROW * x_counter_plastic * COS(PLASTIC_TRAY_ORIENTATION) -50 +200;
		Plastic_Cup_Supply_Position[0] := PLASTIC_CUP_INIT_POSITION [0] - DIST_X_PLASTIC_CENTR_SAME_ROW * x_counter_plastic * COS(PLASTIC_TRAY_ORIENTATION) -50 +200;
		Plastic_Cup_Supply_Above_Pos[1] := PLASTIC_CUP_INIT_POSITION [1] - DIST_Y_PLASTIC_CENTR * y_counter_plastic;
		Plastic_Cup_Supply_Position[1] := PLASTIC_CUP_INIT_POSITION [1] - DIST_Y_PLASTIC_CENTR * y_counter_plastic;
		Plastic_Cups_Remaining := Plastic_Cups_Remaining -1;
		RETURN;
	ELSIF (y_counter_plastic = 3) AND (x_counter_plastic = 7) THEN //this raw has only 5 cups last case
		x_counter_plastic := 0;
		y_counter_plastic := 4;
		Plastic_Cup_Supply_Above_Pos[0] := PLASTIC_CUP_INIT_POSITION [0] - DIST_X_PLASTIC_CENTR_SAME_ROW * x_counter_plastic * COS(PLASTIC_TRAY_ORIENTATION) +200;
		Plastic_Cup_Supply_Position[0] := PLASTIC_CUP_INIT_POSITION [0] - DIST_X_PLASTIC_CENTR_SAME_ROW * x_counter_plastic * COS(PLASTIC_TRAY_ORIENTATION) +200;
		Plastic_Cup_Supply_Above_Pos[1] := PLASTIC_CUP_INIT_POSITION [1] - DIST_Y_PLASTIC_CENTR * y_counter_plastic;
		Plastic_Cup_Supply_Position[1] := PLASTIC_CUP_INIT_POSITION [1] - DIST_Y_PLASTIC_CENTR * y_counter_plastic;
		Plastic_Cups_Remaining := Plastic_Cups_Remaining -1;
		RETURN;
	END_IF

	IF (y_counter_plastic = 4) AND (x_counter_plastic < 8) THEN

		x_counter_plastic := x_counter_plastic + 1;
		Plastic_Cup_Supply_Above_Pos[0] := PLASTIC_CUP_INIT_POSITION [0] - DIST_X_PLASTIC_CENTR_SAME_ROW * x_counter_plastic * COS(PLASTIC_TRAY_ORIENTATION) +200;
		Plastic_Cup_Supply_Position[0] := PLASTIC_CUP_INIT_POSITION [0] - DIST_X_PLASTIC_CENTR_SAME_ROW * x_counter_plastic * COS(PLASTIC_TRAY_ORIENTATION) +200;
		Plastic_Cup_Supply_Above_Pos[1] := PLASTIC_CUP_INIT_POSITION [1] - DIST_Y_PLASTIC_CENTR * y_counter_plastic;
		Plastic_Cup_Supply_Position[1] := PLASTIC_CUP_INIT_POSITION [1] - DIST_Y_PLASTIC_CENTR * y_counter_plastic;
		Plastic_Cups_Remaining := Plastic_Cups_Remaining -1;
		RETURN;
	ELSIF (y_counter_plastic = 4) AND (x_counter_plastic = 8) THEN //this raw has only 5 cups last case
		x_counter_plastic := 0;
		y_counter_plastic := 0;
		Plastic_Cup_Supply_Above_Pos[0] := PLASTIC_CUP_INIT_POSITION [0] - DIST_X_PLASTIC_CENTR_SAME_ROW * x_counter_plastic * COS(PLASTIC_TRAY_ORIENTATION);
		Plastic_Cup_Supply_Position[0] := PLASTIC_CUP_INIT_POSITION [0] - DIST_X_PLASTIC_CENTR_SAME_ROW * x_counter_plastic * COS(PLASTIC_TRAY_ORIENTATION);
		Plastic_Cup_Supply_Above_Pos[1] := PLASTIC_CUP_INIT_POSITION [1] - DIST_Y_PLASTIC_CENTR * y_counter_plastic;
		Plastic_Cup_Supply_Position[1] := PLASTIC_CUP_INIT_POSITION [1] - DIST_Y_PLASTIC_CENTR * y_counter_plastic;
		Plastic_Cups_Remaining := 0;
		RETURN;
	END_IF

	RETURN;

END_FUNCTION
```

#### Paused.st
```iecst
ACTION Paused:

	IF gAssemblyModule.state.stateMachine.stateTransition.resume THEN
		gAssemblyModule.state.stateMachine.operationalState := RUNNING;
	END_IF;

END_ACTION
```

#### Resetting.st
```iecst
ACTION Resetting:
	Mp_Comau.Stop := FALSE;
	IF NOT Mp_Comau.Stopped THEN
		Mp_Parameters.CoordSystem := 0;
		Mp_Parameters.Position := Comau_Resetting_Poition;
		Mp_Comau.MoveDirect := TRUE;
		IF Mp_Comau.MoveDone THEN
			Mp_Comau.MoveDirect := FALSE;
			Mp_Parameters.CoordSystem := 4;
			gAssemblyModule.state.stateMachine.operationalState := IDLE;
		END_IF;
	END_IF
END_ACTION
```

#### Running.st
```iecst
ACTION Running:

END_ACTION
```

#### Stopped.st
```iecst
ACTION Stopped:

	CASE Stopped_Case OF

		GENERAL_STOPPED:

			IF gAssemblyModule.state.stateMachine.stateTransition.reset THEN

				gAssemblyModule.state.stateMachine.operationalState := RESETTING;

			END_IF;

			IF HomeRobot THEN
				Stopped_Case := HOMING_STOPPED;
			END_IF

		HOMING_STOPPED:

			IF DiagCpuIsSimulated() OR  Home_Mode THEN

				FOR i:=0 TO 5 DO
					Mp_JointParameters[i].Homing.Mode := mcHOMING_DIRECT;
					IF i=2 THEN
						Mp_JointParameters[i].Homing.Position := -90;
					ELSE
						Mp_JointParameters[i].Homing.Position := 0;
					END_IF
				END_FOR

			ELSE

				FOR i:=0 TO 5 DO
					Mp_JointParameters[i].Homing.Mode := mcHOMING_DEFAULT;
				END_FOR

			END_IF

			Mp_Comau.Home := TRUE;
			Stopped_Case := EXIT_HOMING_STOPPED;

		EXIT_HOMING_STOPPED:

			IF Mp_Comau.IsHomed AND NOT Mp_Comau.CommandBusy THEN
				Mp_Comau.Home := FALSE;
				Home_Mode := FALSE;
				HomeRobot := FALSE;
				Stopped_Case := GENERAL_STOPPED;
			END_IF

//		MAINTENANCE_STOPPED:
//
//			IF  Assem_PaperTray_Refill_Button THEN
//				Paper_Cups_Remaining := 20;
//			END_IF
//
//			IF Assem_PlasticTray_Refill_Button THEN
//				Plastic_Cups_Remaining := 20;
//				//put position 1 of the trays
//			END_IF
//
//			IF Maintenance_Done THEN
//				Maintenance_Done := FALSE;
//				Stopped_Case := GENERAL_STOPPED;
//				gAssemblyModule.state.stateMachine.operationalState := RESETTING;
//			END_IF

	END_CASE

END_ACTION
```

#### Stopping.st
```iecst
ACTION Stopping:

	gAssemblyModule.skill.goHome.state.stateMachine.stateTransition.abort := TRUE;
	gAssemblyModule.skill.provideCup.state.stateMachine.stateTransition.abort := TRUE;
	gAssemblyModule.skill.providePellet.state.stateMachine.stateTransition.abort := TRUE;

	Mp_Comau.Stop := TRUE;

	IF (gAssemblyModule.skill.goHome.state.stateMachine.operationalState = ABORTED) AND
		(gAssemblyModule.skill.provideCup.state.stateMachine.operationalState = ABORTED) AND
		(gAssemblyModule.skill.providePellet.state.stateMachine.operationalState = ABORTED)	AND
		(Mp_Comau.Stopped) THEN

		gAssemblyModule.state.stateMachine.stateTransition.stop := FALSE;
		Mp_Comau.Stop := FALSE;
		gAssemblyModule.state.stateMachine.operationalState := STOPPED;

	END_IF;

END_ACTION
```

#### Suspended.st
```iecst
ACTION Suspended:
	IF gAssemblyModule.state.stateMachine.stateTransition.unsuspend THEN
		gAssemblyModule.state.stateMachine.operationalState := UNSUSPENDING;

	END_IF;

END_ACTION
```

#### Unholding.st
```iecst
ACTION Unholding:

	gAssemblyModule.state.stateMachine.operationalState := RUNNING;

END_ACTION
```

#### Unsuspending.st
```iecst
ACTION Unsuspending:

		gAssemblyModule.state.stateMachine.operationalState := RUNNING;

END_ACTION
```

#### Clearing.st
```iecst
ACTION Clearing:

	Counter_Clearing_Timeout (IN := TRUE, PT := T#5s);

	IF Counter_Clearing_Timeout.Q THEN
		Event_Code := 100;
		EventLog.Commands.WriteUserEvent := TRUE;
	END_IF;

	CASE Clearing_Case OF

		POWERON:

			//initialize cases
			Stopped_Case := GENERAL_STOPPED;
			provideCup_Case := CUP_SUPPLY_DECISION_CASE;
			providePellet_Case := PELLET_SUPPLY_DECISION_CASE;

			//set safe speed and accel and deccel as default
			Mp_Parameters.Velocity := 1000;
			Mp_Parameters.Deceleration := 10000;
			Mp_Parameters.Acceleration := 10000;

			IF NOT Mp_Comau.PowerOn AND Mp_Comau.Info.ReadyToPowerOn THEN
				Mp_Comau.Power:= TRUE;
				Clearing_Case:= HOMING;
			END_IF

		HOMING:

			IF Mp_Comau.PowerOn THEN

				IF DiagCpuIsSimulated() OR Home_Mode THEN

					FOR i:=0 TO 5 DO
						Mp_JointParameters[i].Homing.Mode := mcHOMING_DIRECT;

						IF i=2 THEN
							Mp_JointParameters[i].Homing.Position := -90;
						ELSE
							Mp_JointParameters[i].Homing.Position := 0;
						END_IF
					END_FOR

				ELSE

					FOR i:=0 TO 5 DO
						Mp_JointParameters[i].Homing.Mode := mcHOMING_DEFAULT;
					END_FOR

				END_IF

				Mp_Comau.Home := TRUE;
				Clearing_Case:= EXIT_CLEARING;

			END_IF

		EXIT_CLEARING:

			IF Mp_Comau.IsHomed AND Mp_Comau.PowerOn AND NOT Mp_Comau.CommandBusy THEN

				Mp_Comau.Home := FALSE;
				Home_Mode := FALSE;
				gAssemblyModule.state.stateMachine.operationalState := STOPPED;
				Clearing_Case:= POWERON;
				Comau_Gripper := FALSE;
				//Disable timer count until next clearing
				IF Counter_Clearing_Timeout.IN THEN
					Counter_Clearing_Timeout (IN := FALSE);
				END_IF;

			END_IF

	END_CASE

END_ACTION
```

#### Completing.st
```iecst
ACTION Completing:
	gAssemblyModule.state.stateMachine.operationalState := COMPLETE;
END_ACTION
```

#### Held.st
```iecst
ACTION Held:

	//Unlock the doors for the refill process
	IF Assem_PaperLock OR Assem_PlasticLock AND NOT Refill_Done THEN
		Assem_PlasticLock := FALSE;
		Assem_PaperLock := FALSE;
	END_IF;

	IF  TON_PlasticDrawer.Q THEN
		Assem_PlasticRemaining := Assem_PlasticTraySize;
		Plastic_RefillDone := TRUE;
	END_IF;

	IF TON_PaperDrawer.Q THEN
		Assem_PaperRemaining := Assem_PaperTraySize;
		Paper_RefillDone := TRUE;
	END_IF;

	IF Refill_Done THEN
		Assem_PlasticLock := TRUE;
		Assem_PaperLock := TRUE;
	END_IF;

	//If everything is closed
	IF Assem_LeftDoorSensor AND Assem_RightDoorSensor AND Assem_PlasticCupsDrawer AND Assem_PaperCupsDrawer
		AND TON_LocksSensor.Q THEN

		Event_Code := 133;
		EventLog.Commands.WriteUserEvent := TRUE;
		//Reset variables to original state
		Refill_Done := FALSE;
		gAssemblyModule.state.stateMachine.operationalState := UNHOLDING;
	END_IF;

	TON_PlasticDrawer(IN := NOT Assem_PlasticCupsDrawer, PT := T#3s);
	TON_PaperDrawer(IN := NOT Assem_PaperCupsDrawer, PT := T#3s);
	TON_LocksSensor(IN := Assem_PaperLock AND Assem_PlasticLock, PT := T#2s);

END_ACTION
```

#### goHome_Aborted.st
```iecst
ACTION goHome_Aborted:

	IF gAssemblyModule.skill.goHome.state.stateMachine.stateTransition.reset THEN
		gAssemblyModule.skill.goHome.state.stateMachine.operationalState := RESETTING;

	ELSIF gAssemblyModule.skill.goHome.state.stateMachine.stateTransition.clear THEN
		gAssemblyModule.skill.goHome.state.stateMachine.operationalState := CLEARING;

	END_IF;

END_ACTION
```

#### goHome_Aborting.st
```iecst
ACTION goHome_Aborting:
//	IF NOT TransitionFromStopped THEN
//		Event_Code := 107;
//		EventLog.Commands.WriteUserEvent := TRUE;
//	END_IF;

	gAssemblyModule.skill.goHome.state.stateMachine.stateTransition.abort 	  := FALSE;
	gAssemblyModule.skill.goHome.state.stateMachine.stateTransition.clear 	  := FALSE;
	gAssemblyModule.skill.goHome.state.stateMachine.stateTransition.hold 	  := FALSE;
	gAssemblyModule.skill.goHome.state.stateMachine.stateTransition.pause 	  := FALSE;
	gAssemblyModule.skill.goHome.state.stateMachine.stateTransition.reset 	  := FALSE;
	gAssemblyModule.skill.goHome.state.stateMachine.stateTransition.resume 	  := FALSE;
	gAssemblyModule.skill.goHome.state.stateMachine.stateTransition.start 	  := FALSE;
	gAssemblyModule.skill.goHome.state.stateMachine.stateTransition.stop 	  := FALSE;
	gAssemblyModule.skill.goHome.state.stateMachine.stateTransition.suspend   := FALSE;
	gAssemblyModule.skill.goHome.state.stateMachine.stateTransition.unhold 	  := FALSE;
	gAssemblyModule.skill.goHome.state.stateMachine.stateTransition.unsuspend := FALSE;

	gAssemblyModule.skill.goHome.state.stateMachine.operationalState := ABORTED;

END_ACTION
```

#### goHome_Holding.st
```iecst
ACTION goHome_Holding:

	gAssemblyModule.skill.goHome.state.stateMachine.operationalState := HELD;

END_ACTION
```

#### goHome_Paused.st
```iecst
ACTION goHome_Paused:

	IF gAssemblyModule.skill.goHome.state.stateMachine.stateTransition.resume THEN
		gAssemblyModule.skill.goHome.state.stateMachine.operationalState := RUNNING;

	END_IF;

END_ACTION
```

#### goHome_Resetting.st
```iecst
ACTION goHome_Resetting:

		gAssemblyModule.skill.goHome.state.stateMachine.operationalState := IDLE;

END_ACTION
```

#### goHome_Running.st
```iecst
ACTION goHome_Running:
	Mp_Parameters.Position := Home_Position;

	Mp_Comau.MoveDirect:=TRUE;
	IF Mp_Comau.MoveDone THEN
		Mp_Comau.MoveDirect := FALSE;
		gAssemblyModule.skill.goHome.state.stateMachine.operationalState := COMPLETING;
	END_IF

END_ACTION
```

#### goHome_Starting.st
```iecst
ACTION goHome_Starting:

	gAssemblyModule.skill.goHome.state.stateMachine.operationalState := RUNNING;

END_ACTION
```

#### goHome_StateErrorReset.st
```iecst
ACTION goHome_StateErrorReset:

	gAssemblyModule.skill.goHome.state.stateMachine.operationalStateError := '';
	gaMessagesModule[57].bMessage_Active := FALSE;

END_ACTION
```

#### goHome_Stopped.st
```iecst
ACTION goHome_Stopped:

	IF gAssemblyModule.skill.goHome.state.stateMachine.stateTransition.reset THEN
		gAssemblyModule.skill.goHome.state.stateMachine.operationalState := RESETTING;
	END_IF;

END_ACTION
```

#### goHome_Suspending.st
```iecst
ACTION goHome_Suspending:

	gAssemblyModule.skill.goHome.state.stateMachine.operationalState := SUSPENDED;

END_ACTION
```

#### goHome_Unholding.st
```iecst
ACTION goHome_Unholding:

		gAssemblyModule.skill.goHome.state.stateMachine.operationalState := RUNNING;

END_ACTION
```

#### goHome_Unsuspending.st
```iecst
ACTION goHome_Unsuspending:

	gAssemblyModule.skill.goHome.state.stateMachine.operationalState := RUNNING;

END_ACTION
```

#### provideCup.st
```iecst
ACTION provideCup:
		(*************************************************************************************************)
		(*************************************************************************************************)
		(* State Machine *)
	CASE gAssemblyModule.skill.provideCup.state.stateMachine.operationalState OF
		(*************************************************************************************************)
		(* RESETTING *)
		RESETTING:
			(*gAssemblyModule.skill.provideCup.state.stateMachine.stateTransition.reset := FALSE;*)

			IF gAssemblyModule.skill.provideCup.state.stateMachine.stateTransition.abort THEN
				gAssemblyModule.skill.provideCup.state.stateMachine.operationalState := ABORTING;

			ELSIF gAssemblyModule.skill.provideCup.state.stateMachine.stateTransition.stop THEN
				gAssemblyModule.skill.provideCup.state.stateMachine.operationalState := STOPPING;

			ELSE
				provideCup_Resetting;

			END_IF;

			(*************************************************************************************************)
			(* IDLE *)
		IDLE:

			gAssemblyModule.skill.provideCup.state.stateMachine.stateTransition.reset := FALSE;

			IF gAssemblyModule.skill.provideCup.state.stateMachine.stateTransition.abort THEN
				gAssemblyModule.skill.provideCup.state.stateMachine.operationalState := ABORTING;

			ELSIF gAssemblyModule.skill.provideCup.state.stateMachine.stateTransition.stop THEN
				gAssemblyModule.skill.provideCup.state.stateMachine.operationalState := STOPPING;

			ELSE
				provideCup_Idle;

			END_IF;

			(*************************************************************************************************)
			(* STARTING *)
		STARTING:
			(*gAssemblyModule.skill.provideCup.state.stateMachine.stateTransition.start := FALSE;*)

			IF gAssemblyModule.skill.provideCup.state.stateMachine.stateTransition.abort THEN
				gAssemblyModule.skill.provideCup.state.stateMachine.operationalState := ABORTING;

			ELSIF gAssemblyModule.skill.provideCup.state.stateMachine.stateTransition.stop THEN
				gAssemblyModule.skill.provideCup.state.stateMachine.operationalState := STOPPING;

			ELSE
				provideCup_Starting;

			END_IF;

			(*************************************************************************************************)
			(* RUNNING *)
		RUNNING:

			gAssemblyModule.skill.provideCup.state.stateMachine.stateTransition.start := FALSE;

			IF gAssemblyModule.skill.provideCup.state.stateMachine.stateTransition.abort THEN
				gAssemblyModule.skill.provideCup.state.stateMachine.operationalState := ABORTING;

			ELSIF gAssemblyModule.skill.provideCup.state.stateMachine.stateTransition.stop THEN
				gAssemblyModule.skill.provideCup.state.stateMachine.operationalState := STOPPING;

			ELSIF gAssemblyModule.skill.provideCup.state.stateMachine.stateTransition.hold THEN
				gAssemblyModule.skill.provideCup.state.stateMachine.operationalState := HOLDING;

			ELSIF gAssemblyModule.skill.provideCup.state.stateMachine.stateTransition.suspend THEN
				//gAssemblyModule.skill.provideCup.state.stateMachine.operationalState := SUSPENDING;

			ELSIF gAssemblyModule.skill.provideCup.state.stateMachine.stateTransition.pause THEN
				//gAssemblyModule.skill.provideCup.state.stateMachine.operationalState := PAUSING;

			ELSE
				provideCup_Running;

			END_IF;

			(*************************************************************************************************)
			(* PAUSING *)
		PAUSING:
			(*	gAssemblyModule.skill.provideCup.state.stateMachine.stateTransition.pause := FALSE;*)

			IF gAssemblyModule.skill.provideCup.state.stateMachine.stateTransition.abort THEN
				gAssemblyModule.skill.provideCup.state.stateMachine.operationalState := ABORTING;

			ELSIF gAssemblyModule.skill.provideCup.state.stateMachine.stateTransition.stop THEN
				gAssemblyModule.skill.provideCup.state.stateMachine.operationalState := STOPPING;

			ELSIF gAssemblyModule.skill.provideCup.state.stateMachine.stateTransition.hold THEN
				//gAssemblyModule.skill.provideCup.state.stateMachine.operationalState := HOLDING;

			ELSIF gAssemblyModule.skill.provideCup.state.stateMachine.stateTransition.suspend THEN
				//gAssemblyModule.skill.provideCup.state.stateMachine.operationalState := SUSPENDING;

			ELSE
				provideCup_Pausing;
			END_IF;

			(*************************************************************************************************)
			(* PAUSED *)
		PAUSED:

			gAssemblyModule.skill.provideCup.state.stateMachine.stateTransition.pause := FALSE;

			IF gAssemblyModule.skill.provideCup.state.stateMachine.stateTransition.abort THEN
				gAssemblyModule.skill.provideCup.state.stateMachine.operationalState := ABORTING;

			ELSIF gAssemblyModule.skill.provideCup.state.stateMachine.stateTransition.stop THEN
				gAssemblyModule.skill.provideCup.state.stateMachine.operationalState := STOPPING;

			ELSIF gAssemblyModule.skill.provideCup.state.stateMachine.stateTransition.hold THEN
				//gAssemblyModule.skill.provideCup.state.stateMachine.operationalState := HOLDING;

			ELSIF gAssemblyModule.skill.provideCup.state.stateMachine.stateTransition.suspend THEN
				//gAssemblyModule.skill.provideCup.state.stateMachine.operationalState := SUSPENDING;

			ELSE
				provideCup_Paused;

			END_IF;

			(*************************************************************************************************)
			(* SUSPENDING *)
		SUSPENDING:
			(*gAssemblyModule.skill.provideCup.state.stateMachine.stateTransition.suspend := FALSE;*)

			IF gAssemblyModule.skill.provideCup.state.stateMachine.stateTransition.abort THEN
				gAssemblyModule.skill.provideCup.state.stateMachine.operationalState := ABORTING;

			ELSIF gAssemblyModule.skill.provideCup.state.stateMachine.stateTransition.stop THEN
				gAssemblyModule.skill.provideCup.state.stateMachine.operationalState := STOPPING;

			ELSIF gAssemblyModule.skill.provideCup.state.stateMachine.stateTransition.hold THEN
				//gAssemblyModule.skill.provideCup.state.stateMachine.operationalState := HOLDING;

			ELSE
				provideCup_Suspending;

			END_IF;

			(*************************************************************************************************)
			(* SUSPENDED *)
		SUSPENDED:

			gAssemblyModule.skill.provideCup.state.stateMachine.stateTransition.suspend := FALSE;

			IF gAssemblyModule.skill.provideCup.state.stateMachine.stateTransition.abort THEN
				gAssemblyModule.skill.provideCup.state.stateMachine.operationalState := ABORTING;

			ELSIF gAssemblyModule.skill.provideCup.state.stateMachine.stateTransition.stop THEN
				gAssemblyModule.skill.provideCup.state.stateMachine.operationalState := STOPPING;

			ELSIF gAssemblyModule.skill.provideCup.state.stateMachine.stateTransition.hold THEN
				//gAssemblyModule.skill.provideCup.state.stateMachine.operationalState := HOLDING;

			ELSE
				provideCup_Suspended;

			END_IF;

			(*************************************************************************************************)
			(* UNSUSPENDING *)
		UNSUSPENDING:
			gAssemblyModule.skill.provideCup.state.stateMachine.stateTransition.unsuspend := FALSE;

			IF gAssemblyModule.skill.provideCup.state.stateMachine.stateTransition.abort THEN
				gAssemblyModule.skill.provideCup.state.stateMachine.operationalState := ABORTING;

			ELSIF gAssemblyModule.skill.provideCup.state.stateMachine.stateTransition.stop THEN
				gAssemblyModule.skill.provideCup.state.stateMachine.operationalState := STOPPING;

			ELSIF gAssemblyModule.skill.provideCup.state.stateMachine.stateTransition.hold THEN
				//gAssemblyModule.skill.provideCup.state.stateMachine.operationalState := HOLDING;

			ELSE
				provideCup_Unsuspending;

			END_IF;

			(*************************************************************************************************)
			(* HOLDING *)
		HOLDING:
			(*gAssemblyModule.skill.provideCup.state.stateMachine.stateTransition.hold := FALSE;*)

			IF gAssemblyModule.state.stateMachine.stateTransition.abort THEN
				gAssemblyModule.state.stateMachine.operationalState := ABORTING;

			ELSIF gAssemblyModule.state.stateMachine.stateTransition.stop THEN
				gAssemblyModule.state.stateMachine.operationalState := STOPPING;

			ELSE
				provideCup_Holding;

			END_IF;

			(*************************************************************************************************)
			(* HELD *)
		HELD:

			gAssemblyModule.skill.provideCup.state.stateMachine.stateTransition.hold := FALSE;

			IF gAssemblyModule.skill.provideCup.state.stateMachine.stateTransition.abort THEN
				gAssemblyModule.skill.provideCup.state.stateMachine.operationalState := ABORTING;

			ELSIF gAssemblyModule.skill.provideCup.state.stateMachine.stateTransition.stop THEN
				gAssemblyModule.skill.provideCup.state.stateMachine.operationalState := STOPPING;

			ELSE
				provideCup_Held;

			END_IF;

			(*************************************************************************************************)
			(* UNHOLDING *)
		UNHOLDING:
			gAssemblyModule.skill.provideCup.state.stateMachine.stateTransition.unhold := FALSE;

			IF gAssemblyModule.skill.provideCup.state.stateMachine.stateTransition.abort THEN
				gAssemblyModule.skill.provideCup.state.stateMachine.operationalState := ABORTING;

			ELSIF gAssemblyModule.skill.provideCup.state.stateMachine.stateTransition.stop THEN
				gAssemblyModule.skill.provideCup.state.stateMachine.operationalState := STOPPING;

			ELSE
				provideCup_Unholding;

			END_IF;

			(*************************************************************************************************)
			(* COMPLETING *)
		COMPLETING:

			IF gAssemblyModule.skill.provideCup.state.stateMachine.stateTransition.abort THEN
				gAssemblyModule.skill.provideCup.state.stateMachine.operationalState := ABORTING;

			ELSIF gAssemblyModule.skill.provideCup.state.stateMachine.stateTransition.stop THEN
				gAssemblyModule.skill.provideCup.state.stateMachine.operationalState := STOPPING;

			ELSE
				provideCup_Completing;

			END_IF;

			(*************************************************************************************************)
			(* COMPLETE *)
		COMPLETE:

			IF gAssemblyModule.skill.provideCup.state.stateMachine.stateTransition.abort THEN
				gAssemblyModule.skill.provideCup.state.stateMachine.operationalState := ABORTING;

			ELSIF gAssemblyModule.skill.provideCup.state.stateMachine.stateTransition.stop THEN
				gAssemblyModule.skill.provideCup.state.stateMachine.operationalState := STOPPING;

			ELSE
				provideCup_Complete;

			END_IF;

			(*************************************************************************************************)
			(* STOPPING *)
		STOPPING:
			(*gAssemblyModule.skill.provideCup.state.stateMachine.stateTransition.stop := FALSE;*)

			IF gAssemblyModule.skill.provideCup.state.stateMachine.stateTransition.abort THEN
				gAssemblyModule.skill.provideCup.state.stateMachine.operationalState := ABORTING;

			ELSE
				provideCup_Stopping;

			END_IF;

			(*************************************************************************************************)
			(* STOPPED *)
		STOPPED:

			gAssemblyModule.skill.provideCup.state.stateMachine.stateTransition.stop := FALSE;

			IF gAssemblyModule.skill.provideCup.state.stateMachine.stateTransition.abort THEN
				gAssemblyModule.skill.provideCup.state.stateMachine.operationalState := ABORTING;

			ELSE
				provideCup_Stopped;

			END_IF;

			(*************************************************************************************************)
			(* ABORTING *)
		ABORTING:
			(*gAssemblyModule.skill.provideCup.state.stateMachine.stateTransition.abort := FALSE;*)

			provideCup_Aborting;

			(*************************************************************************************************)
			(* ABORTED *)
		ABORTED:

			gAssemblyModule.skill.provideCup.state.stateMachine.stateTransition.abort := FALSE;

			provideCup_Aborted;

			(*************************************************************************************************)
			(* CLEARING *)
		CLEARING:
			gAssemblyModule.skill.provideCup.state.stateMachine.stateTransition.clear := FALSE;

			provideCup_Clearing;

			(*************************************************************************************************)
			(* ELSE *)
		ELSE;

	END_CASE;
END_ACTION
```

#### provideCup_Aborted.st
```iecst
ACTION provideCup_Aborted:

	IF gAssemblyModule.skill.provideCup.state.stateMachine.stateTransition.reset THEN
		gAssemblyModule.skill.provideCup.state.stateMachine.operationalState := RESETTING;

	ELSIF gAssemblyModule.skill.provideCup.state.stateMachine.stateTransition.clear THEN
		gAssemblyModule.skill.provideCup.state.stateMachine.operationalState := CLEARING;

	END_IF;

END_ACTION
```

#### provideCup_Aborting.st
```iecst
ACTION provideCup_Aborting:

	gAssemblyModule.skill.provideCup.state.stateMachine.stateTransition.abort 	  := FALSE;
	gAssemblyModule.skill.provideCup.state.stateMachine.stateTransition.clear 	  := FALSE;
	gAssemblyModule.skill.provideCup.state.stateMachine.stateTransition.hold 	  := FALSE;
	gAssemblyModule.skill.provideCup.state.stateMachine.stateTransition.pause 	  := FALSE;
	gAssemblyModule.skill.provideCup.state.stateMachine.stateTransition.reset 	  := FALSE;
	gAssemblyModule.skill.provideCup.state.stateMachine.stateTransition.resume 	  := FALSE;
	gAssemblyModule.skill.provideCup.state.stateMachine.stateTransition.start 	  := FALSE;
	gAssemblyModule.skill.provideCup.state.stateMachine.stateTransition.stop 	  := FALSE;
	gAssemblyModule.skill.provideCup.state.stateMachine.stateTransition.suspend   := FALSE;
	gAssemblyModule.skill.provideCup.state.stateMachine.stateTransition.unhold 	  := FALSE;
	gAssemblyModule.skill.provideCup.state.stateMachine.stateTransition.unsuspend := FALSE;

	//jump one cup in case General SM goes to stopped or aborted
	IF  gAssemblyModule.skill.provideCup.inputParameters.cupType = 1 THEN	// 1 = Paper
			x_counter_paper := x_counter_paper +1;
			Assem_PaperRemaining := Assem_PaperRemaining -1;
	ELSIF gAssemblyModule.skill.provideCup.inputParameters.cupType = 2 THEN	// 2 = Plastic
			x_counter_plastic := x_counter_plastic +1;
			Assem_PlasticRemaining := Assem_PlasticRemaining -1;
	END_IF

	gAssemblyModule.skill.provideCup.state.stateMachine.operationalState := ABORTED;

END_ACTION
```

#### provideCup_Clearing.st
```iecst
ACTION provideCup_Clearing:

	gAssemblyModule.skill.provideCup.state.stateMachine.stateTransition.clear := FALSE;

	gAssemblyModule.skill.provideCup.state.stateMachine.operationalState := STOPPED;

END_ACTION
```

#### provideCup_Completing.st
```iecst
ACTION provideCup_Completing:

	provideCup_Case := CUP_SUPPLY_DECISION_CASE;

	gAssemblyModule.skill.provideCup.OutputParameters.SecondOutputParam := Assem_PlasticRemaining;
	gAssemblyModule.skill.provideCup.OutputParameters.FirstOutputParam := Assem_PaperRemaining;

	gAssemblyModule.skill.provideCup.inputParameters.cupType := 0;

	gAssemblyModule.skill.provideCup.state.stateMachine.operationalState := COMPLETE;

END_ACTION
```

#### provideCup_Holding.st
```iecst
ACTION provideCup_Holding:

	gAssemblyModule.skill.provideCup.state.stateMachine.operationalState := HELD;

END_ACTION
```

#### provideCup_Running.st
```iecst
ACTION provideCup_Running:

	IF (Assem_PaperRemaining = 0 AND gAssemblyModule.skill.provideCup.inputParameters.cupType = 1 ) AND NOT Checked THEN
		Event_Code := 130;
		EventLog.Commands.WriteUserEvent := TRUE;

	ELSIF (Assem_PlasticRemaining = 0 AND gAssemblyModule.skill.provideCup.inputParameters.cupType = 2 ) AND NOT Checked THEN
		Event_Code := 130;
		EventLog.Commands.WriteUserEvent := TRUE;

	ELSIF Checked THEN
		CASE provideCup_Case OF

			CUP_SUPPLY_DECISION_CASE:

				IF  gAssemblyModule.skill.provideCup.inputParameters.cupType = 1 THEN	// 1 = Paper

					IF Assem_PaperRemaining > 0 THEN
						provideCup_Case := PAPER_CUP_SAFE_POSITION_CASE;
					ELSE
						provideCup_Case := CUP_SUPPLY_FINAL_CASE1;
						Event_Code := 132;
						EventLog.Commands.WriteUserEvent := TRUE;
					END_IF

				ELSIF gAssemblyModule.skill.provideCup.inputParameters.cupType = 2 THEN	// 2 = Plastic

					IF Assem_PlasticRemaining > 0 THEN
						provideCup_Case := PLASTIC_CUP_SAFE_POSITION_CASE;
					ELSE
						provideCup_Case := CUP_SUPPLY_FINAL_CASE1;
						Event_Code := 132;
						EventLog.Commands.WriteUserEvent := TRUE;
					END_IF

				ELSE

					provideCup_Case := CUP_SUPPLY_FINAL_CASE1;

				END_IF;

				////////////////////////////////////////////////////////////////////////////////////////////////////

			PLASTIC_CUP_SAFE_POSITION_CASE:

				Mp_Parameters.Position := Plastic_Cup_Safe_Pos;
				Mp_Comau.MoveLinear :=TRUE;
				IF Mp_Comau.MoveDone THEN
					Mp_Comau.MoveLinear := FALSE;
					provideCup_Case := PLASTIC_CUP_ABOVE_POSITION_CASE;
				END_IF;

			PLASTIC_CUP_ABOVE_POSITION_CASE:

				Mp_Parameters.Position := Plastic_Cup_Supply_Above_Pos;
				Mp_Comau.MoveLinear :=TRUE;
				IF Mp_Comau.MoveDone THEN
					Mp_Comau.MoveLinear := FALSE;
					provideCup_Case := PLASTIC_CUP_POSITION_CASE;
				END_IF;

			PLASTIC_CUP_POSITION_CASE:

				Mp_Parameters.Position := Plastic_Cup_Supply_Position;
				Mp_Comau.MoveLinear := TRUE;

				IF Mp_Comau.MoveDone THEN
					Mp_Comau.MoveLinear := FALSE;
					Comau_Gripper := TRUE;
					provideCup_Case := PLASTIC_CUP_TIMER_CASE;
				END_IF;

			PLASTIC_CUP_TIMER_CASE:

				Counter_GrabbingCups_Timeout(IN := TRUE, PT := T#0.5s);

				//If the clearing takes more time than expected the supertrak goes into aborted
				IF Counter_GrabbingCups_Timeout.Q THEN
					Counter_GrabbingCups_Timeout(IN := FALSE);
					provideCup_Case := PLASTIC_CUP_ABOVE_POSITION_CASE1;
				END_IF;

			PLASTIC_CUP_ABOVE_POSITION_CASE1:

				Mp_Parameters.Position := Plastic_Cup_Supply_Above_Pos;
				Mp_Comau.MoveLinear := TRUE;
				IF Mp_Comau.MoveDone THEN
					Mp_Comau.MoveLinear := FALSE;
					provideCup_Case := PLASTIC_CUP_SAFE_POSITION_CASE1;
				END_IF;

			PLASTIC_CUP_SAFE_POSITION_CASE1:

				Mp_Parameters.Position := Plastic_Cup_Safe_Pos;
				Mp_Comau.MoveLinear := TRUE;
				IF Mp_Comau.MoveDone THEN
					Mp_Comau.MoveLinear := FALSE;
					provideCup_Case := SUPERTRAK_ABOVE_POSITION_CASE;
				END_IF;

				//////////////////////////////////////////////////////////////////////////////////////////////////

			PAPER_CUP_SAFE_POSITION_CASE:

				Mp_Parameters.Position := Paper_Cup_Safe_Pos;
				Mp_Comau.MoveLinear :=TRUE;
				IF Mp_Comau.MoveDone THEN
					Mp_Comau.MoveLinear := FALSE;
					provideCup_Case := PAPER_CUP_ABOVE_POSITION_CASE;
				END_IF;

			PAPER_CUP_ABOVE_POSITION_CASE:

				Mp_Parameters.Position := Paper_Cup_Supply_Above_Pos;
				Mp_Comau.MoveLinear :=TRUE;
				IF Mp_Comau.MoveDone THEN
					Mp_Comau.MoveLinear := FALSE;
					Comau_Gripper := TRUE;
					provideCup_Case := PAPER_CUP_POSITION_CASE;
				END_IF;

			PAPER_CUP_POSITION_CASE:

				Mp_Parameters.Position := Paper_Cup_Supply_Position;
				Mp_Comau.MoveLinear := TRUE;
				IF Mp_Comau.MoveDone THEN
					Mp_Comau.MoveLinear := FALSE;
					provideCup_Case := PAPER_CUP_TIMER_CASE;
				END_IF;

			PAPER_CUP_TIMER_CASE:

				Counter_GrabbingCups_Timeout(IN := TRUE, PT := T#0.5s);

				//If the clearing takes more time than expected the supertrak goes into aborted
				IF Counter_GrabbingCups_Timeout.Q THEN
					Counter_GrabbingCups_Timeout(IN := FALSE);
					provideCup_Case := PAPER_CUP_ABOVE_POSITION_CASE1;
				END_IF;

			PAPER_CUP_ABOVE_POSITION_CASE1:

				Mp_Parameters.Position := Paper_Cup_Supply_Above_Pos;
				Mp_Comau.MoveLinear := TRUE;
				IF Mp_Comau.MoveDone THEN
					Mp_Comau.MoveLinear := FALSE;
					provideCup_Case := PAPER_CUP_SAFE_POSITION_CASE1;
				END_IF;

			PAPER_CUP_SAFE_POSITION_CASE1:

				Mp_Parameters.Position := Paper_Cup_Safe_Pos;
				Mp_Comau.MoveLinear := TRUE;
				IF Mp_Comau.MoveDone THEN
					Mp_Comau.MoveLinear := FALSE;
					provideCup_Case := SUPERTRAK_ABOVE_POSITION_CASE;
				END_IF;

				/////////////////////////////////////////////////////////////////////////////////////////////////////////////

			SUPERTRAK_ABOVE_POSITION_CASE:

				Mp_Parameters.Position := Supertrak_Above_Position;
				Mp_Comau.MoveLinear := TRUE;
				IF Mp_Comau.MoveDone THEN
					Mp_Comau.MoveLinear := FALSE;
					provideCup_Case := SUPERTRAK_POSITION_CASE;
				END_IF;

			SUPERTRAK_POSITION_CASE:

				Mp_Parameters.Position := Supertrak_Position;
				Mp_Comau.MoveLinear := TRUE;
				IF Mp_Comau.MoveDone THEN
					Mp_Comau.MoveLinear := FALSE;
					Comau_Gripper := FALSE;								//IP variable
					provideCup_Case := SUPERTRAK_TIMER_CASE;
				END_IF;

			SUPERTRAK_TIMER_CASE:

				Counter_LeavingCups_Timeout(IN := TRUE, PT := T#0.5s);

				//If the clearing takes more time than expected the supertrak goes into aborted
				IF Counter_LeavingCups_Timeout.Q THEN
					Counter_LeavingCups_Timeout(IN := FALSE);
					provideCup_Case := SUPERTRAK_ABOVE_POSITION_CASE1;
				END_IF;

			SUPERTRAK_ABOVE_POSITION_CASE1:

				Mp_Parameters.Position := Supertrak_Above_Position;
				Mp_Comau.MoveLinear := TRUE;
				IF Mp_Comau.MoveDone THEN
					Mp_Comau.MoveLinear := FALSE;
					provideCup_Case := SAFE_POSITION_CASE;
				END_IF;

			SAFE_POSITION_CASE:

				Mp_Parameters.Position := Home_Position;
				Mp_Comau.MoveLinear:=TRUE;
				IF Mp_Comau.MoveDone THEN
					Mp_Comau.MoveLinear := FALSE;
					provideCup_Case := CUP_SUPPLY_FINAL_CASE;
				END_IF;

			CUP_SUPPLY_FINAL_CASE:

				IF  gAssemblyModule.skill.provideCup.inputParameters.cupType = 1 THEN	// 1 = Paper
					F_Paper_Update_Positions(
						PAPER_CUP_INIT_POSITION,
						PAPER_TRAY_ORIENTATION,
						DIST_X_PAPER_CENTR_SAME_ROW,
						DIST_X_PAPER_CENTR_DIFF_ROW,
						DIST_Y_PAPER_CENTR,
						Paper_Cup_Supply_Above_Pos,
						Paper_Cup_Supply_Position,
						x_counter_paper,
						y_counter_paper,
						Assem_PaperRemaining);
				ELSIF gAssemblyModule.skill.provideCup.inputParameters.cupType = 2 THEN	// 2 = Plastic
					F_Plastic_Update_Positions(
						PLASTIC_CUP_INIT_POSITION,
						PLASTIC_TRAY_ORIENTATION,
						DIST_X_PLASTIC_CENTR_SAME_ROW,
						DIST_X_PLASTIC_CENTR_DIFF_ROW,
						DIST_Y_PLASTIC_CENTR,
						Plastic_Cup_Supply_Above_Pos,
						Plastic_Cup_Supply_Position,
						x_counter_plastic,
						y_counter_plastic,
						Assem_PlasticRemaining);
				END_IF

				provideCup_Case := CUP_SUPPLY_FINAL_CASE1;

			CUP_SUPPLY_FINAL_CASE1:

				gAssemblyModule.skill.provideCup.state.stateMachine.operationalState := COMPLETING;
				//provideCup_Case := Cup_Supply_Decision_Case;

			ELSE
				;

		END_CASE;
	ELSE
		Checked := TRUE;
	END_IF;

END_ACTION
```

#### provideCup_Starting.st
```iecst
ACTION provideCup_Starting:

	gAssemblyModule.skill.provideCup.state.stateMachine.operationalState := RUNNING;

END_ACTION
```

#### provideCup_Stopped.st
```iecst
ACTION provideCup_Stopped:

	IF gAssemblyModule.skill.provideCup.state.stateMachine.stateTransition.reset THEN
		gAssemblyModule.skill.provideCup.state.stateMachine.operationalState := RESETTING;
	END_IF;

END_ACTION
```

#### provideCup_Stopping.st
```iecst
ACTION provideCup_Stopping:

	gAssemblyModule.skill.provideCup.state.stateMachine.operationalState := STOPPED;

END_ACTION
```

#### provideCup_Suspending.st
```iecst
ACTION provideCup_Suspending:

	gAssemblyModule.skill.provideCup.state.stateMachine.operationalState := SUSPENDED;

END_ACTION
```

#### provideCup_Unholding.st
```iecst
ACTION provideCup_Unholding:

		gAssemblyModule.skill.provideCup.state.stateMachine.operationalState := RUNNING;

END_ACTION
```
